(* alternatively
Sched.nDefaultValue										:= E_BA_BuildingMode.eDefault;
Sched.bWriteWeekly										:= FALSE;
//	Monday
Sched.aWeek[E_BA_Weekday.eMonday,1].eState				:= E_BA_SchedEntryState.eValue;
Sched.aWeek[E_BA_Weekday.eMonday,1].uValue.udiVal		:= E_BA_BuildingMode.eCleaning;
Sched.aWeek[E_BA_Weekday.eMonday,1].stTime.nHour		:= 19;
Sched.aWeek[E_BA_Weekday.eMonday,1].stTime.nMinute		:= 0;
Sched.aWeek[E_BA_Weekday.eMonday,1].stTime.nSecond		:= 0;
Sched.aWeek[E_BA_Weekday.eMonday,2].eState				:= E_BA_SchedEntryState.eValue;
Sched.aWeek[E_BA_Weekday.eMonday,2].uValue.udiVal		:= E_BA_BuildingMode.eNightWatch;
Sched.aWeek[E_BA_Weekday.eMonday,2].stTime.nHour		:= 20;
Sched.aWeek[E_BA_Weekday.eMonday,2].stTime.nMinute		:= 0;
Sched.aWeek[E_BA_Weekday.eMonday,2].stTime.nSecond		:= 0;
Sched.aWeek[E_BA_Weekday.eMonday,3].eState				:= E_BA_SchedEntryState.eValue;
Sched.aWeek[E_BA_Weekday.eMonday,3].uValue.udiVal		:= E_BA_BuildingMode.eDefault;
Sched.aWeek[E_BA_Weekday.eMonday,3].stTime.nHour		:= 0;
Sched.aWeek[E_BA_Weekday.eMonday,3].stTime.nMinute		:= 0;
Sched.aWeek[E_BA_Weekday.eMonday,3].stTime.nSecond		:= 0;
//	Tuesday
Sched.aWeek[E_BA_Weekday.eTuesday,1].eState				:= E_BA_SchedEntryState.eValue;
Sched.aWeek[E_BA_Weekday.eTuesday,1].uValue.udiVal		:= E_BA_BuildingMode.eCleaning;
Sched.aWeek[E_BA_Weekday.eTuesday,1].stTime.nHour		:= 19;
Sched.aWeek[E_BA_Weekday.eTuesday,1].stTime.nMinute		:= 0;
Sched.aWeek[E_BA_Weekday.eTuesday,1].stTime.nSecond		:= 0;
Sched.aWeek[E_BA_Weekday.eTuesday,2].eState				:= E_BA_SchedEntryState.eValue;
Sched.aWeek[E_BA_Weekday.eTuesday,2].uValue.udiVal		:= E_BA_BuildingMode.eNightWatch;
Sched.aWeek[E_BA_Weekday.eTuesday,2].stTime.nHour		:= 20;
Sched.aWeek[E_BA_Weekday.eTuesday,2].stTime.nMinute		:= 0;
Sched.aWeek[E_BA_Weekday.eTuesday,2].stTime.nSecond		:= 0;
Sched.aWeek[E_BA_Weekday.eTuesday,3].eState				:= E_BA_SchedEntryState.eValue;
Sched.aWeek[E_BA_Weekday.eTuesday,3].uValue.udiVal		:= E_BA_BuildingMode.eDefault;
Sched.aWeek[E_BA_Weekday.eTuesday,3].stTime.nHour		:= 0;
Sched.aWeek[E_BA_Weekday.eTuesday,3].stTime.nMinute		:= 0;
Sched.aWeek[E_BA_Weekday.eTuesday,3].stTime.nSecond		:= 0;
//	Wednesday
Sched.aWeek[E_BA_Weekday.eWednesday,1].eState			:= E_BA_SchedEntryState.eValue;
Sched.aWeek[E_BA_Weekday.eWednesday,1].uValue.udiVal	:= E_BA_BuildingMode.eCleaning;
Sched.aWeek[E_BA_Weekday.eWednesday,1].stTime.nHour		:= 19;
Sched.aWeek[E_BA_Weekday.eWednesday,1].stTime.nMinute	:= 0;
Sched.aWeek[E_BA_Weekday.eWednesday,1].stTime.nSecond	:= 0;
Sched.aWeek[E_BA_Weekday.eWednesday,2].eState			:= E_BA_SchedEntryState.eValue;
Sched.aWeek[E_BA_Weekday.eWednesday,2].uValue.udiVal	:= E_BA_BuildingMode.eNightWatch;
Sched.aWeek[E_BA_Weekday.eWednesday,2].stTime.nHour		:= 20;
Sched.aWeek[E_BA_Weekday.eWednesday,2].stTime.nMinute	:= 0;
Sched.aWeek[E_BA_Weekday.eWednesday,2].stTime.nSecond	:= 0;
Sched.aWeek[E_BA_Weekday.eWednesday,3].eState			:= E_BA_SchedEntryState.eValue;
Sched.aWeek[E_BA_Weekday.eWednesday,3].uValue.udiVal	:= E_BA_BuildingMode.eDefault;
Sched.aWeek[E_BA_Weekday.eWednesday,3].stTime.nHour		:= 0;
Sched.aWeek[E_BA_Weekday.eWednesday,3].stTime.nMinute	:= 0;
Sched.aWeek[E_BA_Weekday.eWednesday,3].stTime.nSecond	:= 0;
//	Thursday
Sched.aWeek[E_BA_Weekday.eThursday,1].eState			:= E_BA_SchedEntryState.eValue;
Sched.aWeek[E_BA_Weekday.eThursday,1].uValue.udiVal		:=E_BA_BuildingMode.eCleaning;
Sched.aWeek[E_BA_Weekday.eThursday,1].stTime.nHour		:= 19;
Sched.aWeek[E_BA_Weekday.eThursday,1].stTime.nMinute	:= 0;
Sched.aWeek[E_BA_Weekday.eThursday,1].stTime.nSecond	:= 0;
Sched.aWeek[E_BA_Weekday.eThursday,2].eState			:= E_BA_SchedEntryState.eValue;
Sched.aWeek[E_BA_Weekday.eThursday,2].uValue.udiVal		:= E_BA_BuildingMode.eNightWatch;
Sched.aWeek[E_BA_Weekday.eThursday,2].stTime.nHour		:= 20;
Sched.aWeek[E_BA_Weekday.eThursday,2].stTime.nMinute	:= 0;
Sched.aWeek[E_BA_Weekday.eThursday,2].stTime.nSecond	:= 0;
Sched.aWeek[E_BA_Weekday.eThursday,3].eState			:= E_BA_SchedEntryState.eValue;
Sched.aWeek[E_BA_Weekday.eThursday,3].uValue.udiVal		:= E_BA_BuildingMode.eDefault;
Sched.aWeek[E_BA_Weekday.eThursday,3].stTime.nHour		:= 0;
Sched.aWeek[E_BA_Weekday.eThursday,3].stTime.nMinute	:= 0;
Sched.aWeek[E_BA_Weekday.eThursday,3].stTime.nSecond	:= 0;
//	Friday
Sched.aWeek[E_BA_Weekday.eFriday,1].eState				:= E_BA_SchedEntryState.eValue;
Sched.aWeek[E_BA_Weekday.eFriday,1].uValue.udiVal		:= E_BA_BuildingMode.eCleaning;
Sched.aWeek[E_BA_Weekday.eFriday,1].stTime.nHour		:= 19;
Sched.aWeek[E_BA_Weekday.eFriday,1].stTime.nMinute		:= 0;
Sched.aWeek[E_BA_Weekday.eFriday,1].stTime.nSecond		:= 0;
Sched.aWeek[E_BA_Weekday.eFriday,2].eState				:= E_BA_SchedEntryState.eValue;
Sched.aWeek[E_BA_Weekday.eFriday,2].uValue.udiVal		:= E_BA_BuildingMode.eNightWatch;
Sched.aWeek[E_BA_Weekday.eFriday,2].stTime.nHour		:= 20;
Sched.aWeek[E_BA_Weekday.eFriday,2].stTime.nMinute		:= 0;
Sched.aWeek[E_BA_Weekday.eFriday,2].stTime.nSecond		:= 0;
Sched.aWeek[E_BA_Weekday.eFriday,3].eState				:= E_BA_SchedEntryState.eValue;
Sched.aWeek[E_BA_Weekday.eFriday,3].uValue.udiVal		:= E_BA_BuildingMode.eDefault;
Sched.aWeek[E_BA_Weekday.eFriday,3].stTime.nHour		:= 0;
Sched.aWeek[E_BA_Weekday.eFriday,3].stTime.nMinute		:= 0;
Sched.aWeek[E_BA_Weekday.eFriday,3].stTime.nSecond		:= 0; 
*)
END_METHOD

END_FUNCTION_BLOCK

// ---- Templates/POUs/Trade/BuildingAutomation/GlobalEventsAndSettings/FB_BA_WeatherParameter.TcPOU
{region '#Template'}
	{attribute 'Version' := '5.0.0.0'}
	{attribute 'Tags' := '"LCID": "1031", "Text": "General, Settings, Parameters, Basics"'}
	{attribute 'Tags' := '"LCID": "1033", "Text": "General, Settings, Parameters, Basics"'}
	{attribute 'Using' := '"Type": "Template", "URI": "BA2_Param"'}
	{attribute 'Description' := '"LCID": "1031", "Text": "Witterungsparameter für die Templates"'}
	{attribute 'Description' := '"LCID": "1033", "Text": "Weather parameters for the templates"'}
{endregion}
FUNCTION_BLOCK FB_BA_WeatherParameter EXTENDS FB_BA_View
VAR_INPUT
	fTWth					: REAL;	//	Weather temperature
END_VAR
VAR_OUTPUT
	fSpFrstProtec			: REAL;  // frost protection setpoint. for eg. Heating circutis in protection mode
	fTWthLowLimit			: REAL;  // below this value all frostprotection funcktions in HVAC-Plants will be enabled
	bTWthLowLimit			: BOOL;  // is TRUE when the outside temperature is below the value from fTWthLowLimit 
	fTWthDamped				: REAL;  // damped outside temperature
	bTWthDampedLowLimit		: BOOL;	
END_VAR
VAR_INPUT CONSTANT
	SpFrstProtec			: FB_BA_AV_Op;		
	TWthLowLimitVal			: FB_BA_AV_Op;																
	TWthLowLimit			: FB_BA_BV_Op;								
	TWthDamped				: FB_BA_AV_Op;		
	TWthDampedLowLimit		: FB_BA_BV_Op;	
END_VAR
VAR
	TWthLowLimitHys			: FB_BA_Swi2P;
	Average					: FB_BA_TiAvrg;
	TWthDampedLowLimitHys	: FB_BA_Swi2P;
END_VAR

SUPER^(); // FB_BA_View
SpFrstProtec(); // FB_BA_AV_Op
fSpFrstProtec := SpFrstProtec.fPresentValue;
TWthLowLimitVal(); // FB_BA_AV_Op
fTWthLowLimit := TWthLowLimitVal.fPresentValue;
TWthLowLimitHys(bEn := TRUE, fIn := fTWth, fOn := fTWthLowLimit, fOff := fTWthLowLimit + 1); // FB_BA_Swi2P
TWthLowLimit(bValuePgm := TWthLowLimitHys.bQ); // FB_BA_BV_Op
bTWthLowLimit := TWthLowLimit.bPresentValue;
Average(bEn := BA2_Param.bDlyStartPLC, fIn := fTWth, nIntval := 900, nNumOfElem := 96); // FB_BA_TiAvrg
TWthDamped(fValuePgm := Average.fOut); // FB_BA_AV_Op
fTWthDamped := TWthDamped.fPresentValue;
TWthDampedLowLimitHys(bEn := TRUE, fIn := fTWthDamped, fOn := fTWthLowLimit, fOff := fTWthLowLimit + 1.0); // FB_BA_Swi2P
TWthDampedLowLimit(bValuePgm := TWthDampedLowLimitHys.bQ); // FB_BA_BV_Op
bTWthDampedLowLimit := TWthDampedLowLimit.bPresentValue;

METHOD FB_init : BOOL
VAR_INPUT
	bInitRetains : BOOL; // if TRUE, the retain variables are initialized (warm start / cold start)
	bInCopyCode : BOOL;  // if TRUE, the instance afterwards gets moved into the copy code (online change)
END_VAR
SpFrstProtec.iParent				:= THIS^;
SpFrstProtec.iLabel					:= LblCtl_SetpointFrostProtection;
SpFrstProtec.eUnit					:= E_BA_Unit.eTemperature_DegreesCelsius;  
SpFrstProtec.fValueRm				:= 5.0;
SpFrstProtec.fCOVIncrement			:= BA2_Param.fDefCOVIncrement;							

TWthLowLimitVal.iParent				:= THIS^;
TWthLowLimitVal.iLabel				:= LblCtl_SetpointMinimumOutsideTemperature;
TWthLowLimitVal.eUnit				:= E_BA_Unit.eTemperature_DegreesCelsius;  
TWthLowLimitVal.fValueRm			:= 8.0;
TWthLowLimitVal.fCOVIncrement		:= BA2_Param.fDefCOVIncrement;							

TWthLowLimit.iParent				:= THIS^;	
TWthLowLimit.iLabel					:= LblCtl_OperationalMessageTemperatureWeatherLowLimit;
TWthLowLimit.sInactiveText			:= txtEvent_Off;
TWthLowLimit.sActiveText			:= txtEvent_On;
TWthLowLimit.bValueRm				:= FALSE;		
TWthLowLimit.eToggleMode 			:= E_BA_ToggleMode.eSwitch;

TWthDamped.iParent					:= THIS^;
TWthDamped.iLabel					:= LblCtl_MeanDamped;
TWthDamped.eUnit					:= E_BA_Unit.eTemperature_DegreesCelsius;  
TWthDamped.fValueRm					:= 0.0;
TWthDamped.fCOVIncrement			:= BA2_Param.fDefCOVIncrement;							

TWthDampedLowLimit.iParent			:= THIS^;	
TWthDampedLowLimit.iLabel			:= LblCtl_OperationalMessageTemperatureWeatherDampedLowLimit;	
TWthDampedLowLimit.sInactiveText	:= txtEvent_Off;
TWthDampedLowLimit.sActiveText		:= txtEvent_On;
TWthDampedLowLimit.bValueRm			:= FALSE;								
TWthDampedLowLimit.eToggleMode 		:= E_BA_ToggleMode.eSwitch;
END_METHOD

END_FUNCTION_BLOCK

// ---- Templates/POUs/Trade/BuildingAutomation/WeatherStation/FB_BA_WeatherStation_Draft.TcPOU
{region '#Template'}
	{attribute 'Version' := '5.0.1.0'}
	{attribute 'Tags' := '"LCID": "1031", "Text": "Plant, Weatherstation, Draft"'}
	{attribute 'Tags' := '"LCID": "1033", "Text": "Plant, Weatherstation, Draft"'}
	{attribute 'Using' := '"Type": "Template", "URI": "LblComp"'}		 		 
	{attribute 'Description' := '"LCID": "1031", "Text": "Vorlage-Template: beinhaltet alle Objekte, die Eingangsverknüpfung zu diesen muss vom Anwender erstellt werden"'}
	{attribute 'Description' := '"LCID": "1033", "Text": "Draft-template: contains all objects to be connected to appropriate inputs by the user"'}
{endregion}
FUNCTION_BLOCK FB_BA_WeatherStation_Draft EXTENDS FB_BA_View
VAR_INPUT CONSTANT
	Dstb						: FB_BA_BI;
	Rain						: FB_BA_BI;
	WthT						: FB_BA_AI;
	DewPtT						: FB_BA_AI; 
	PrssAbs						: FB_BA_AI;
	PrssRel						: FB_BA_AI;
	HumAbs						: FB_BA_AI;
	HumRel						: FB_BA_AI;
	Brightness_N				: FB_BA_AI;
	Brightness_S				: FB_BA_AI;
	Brightness_E				: FB_BA_AI;
	Brightness_W				: FB_BA_AI;
	Dawn						: FB_BA_AI;
	GlobRadn					: FB_BA_AI;      
	WndDir						: FB_BA_AI;
	WndSpd						: FB_BA_AI; 
	Latd						: FB_BA_AI;  
	Lngt						: FB_BA_AI; 
	SunAzm						: FB_BA_AI;
	SunElv						: FB_BA_AI;                 
END_VAR	

VAR
	stDateTime_PLACEHOLDER		: TIMESTRUCT;			// Placeholder-variable, so the template can be compiled correctly
														// to be replaced by an appropriate timestruct
END_VAR

SUPER^(); // FB_BA_View
Dstb(); // FB_BA_BI
Site.stWeatherStation.bDisturb := Dstb.bPresentValue;
Rain(); // FB_BA_BI
Site.stWeatherStation.bRain := Rain.bPresentValue;
WndSpd(); // FB_BA_AI
Site.stWeatherStation.fWindSpeed := WndSpd.fPresentValue;
WthT(); // FB_BA_AI
Site.stWeatherStation.fOutsideTemperature := WthT.fPresentValue;
DewPtT(); // FB_BA_AI
Site.stWeatherStation.fDewPointTemperature := DewPtT.fPresentValue;
PrssAbs(); // FB_BA_AI
Site.stWeatherStation.fPressureAbs := PrssAbs.fPresentValue;
PrssRel(); // FB_BA_AI
Site.stWeatherStation.fPressureRel := PrssRel.fPresentValue;
Dawn(); // FB_BA_AI
Site.stWeatherStation.fDawn := Dawn.fPresentValue;
GlobRadn(); // FB_BA_AI
Site.stWeatherStation.fGlobalRadiation := GlobRadn.fPresentValue;
WndDir(); // FB_BA_AI
Site.stWeatherStation.fWindDirection := WndDir.fPresentValue;
HumAbs(); // FB_BA_AI
Site.stWeatherStation.fHumidityAbs := HumAbs.fPresentValue;
HumRel(); // FB_BA_AI
Site.stWeatherStation.fHumidityRel := HumRel.fPresentValue;
Latd(); // FB_BA_AI
Site.stWeatherStation.fLatitude := Latd.fPresentValue;
Lngt(); // FB_BA_AI
Site.stWeatherStation.fLongitude := Lngt.fPresentValue;
SunAzm(); // FB_BA_AI
Site.stWeatherStation.fSunAzimuth := SunAzm.fPresentValue;
SunElv(); // FB_BA_AI
Site.stWeatherStation.fSunElevation := SunElv.fPresentValue;
Brightness_N(); // FB_BA_AI
Site.stWeatherStation.fBrightnessNorth := Brightness_N.fPresentValue;
Brightness_S(); // FB_BA_AI
Site.stWeatherStation.fBrightnessSouth := Brightness_S.fPresentValue;
Brightness_E(); // FB_BA_AI
Site.stWeatherStation.fBrightnessEast := Brightness_E.fPresentValue;
Brightness_W(); // FB_BA_AI
Site.stWeatherStation.fBrightnessWest := Brightness_W.fPresentValue;
Site.stWeatherStation.stDateTime := stDateTime_PLACEHOLDER;

METHOD FB_init : BOOL
VAR_INPUT
	bInitRetains : BOOL; // if TRUE, the retain variables are initialized (warm start / cold start)
	bInCopyCode : BOOL;  // if TRUE, the instance afterwards gets moved into the copy code (online change)
END_VAR
Dstb.iParent							:= THIS^;
Dstb.iLabel								:= LblComp_Wth_WeatherStation; 	
Dstb.sActiveText 						:= txtEvent_Yes;
Dstb.sInactiveText 						:= txtEvent_No;
Dstb.nEventClassID						:= EC_ID.NC60;
Dstb.aEventTransitionText[1]			:= txtEvent_No;
Dstb.aEventTransitionText[2]			:= txtEvent_None;
Dstb.aEventTransitionText[3]			:= txtEvent_Yes;
Dstb.bEventDetectionEnable				:= FALSE;	  
						
Rain.iParent							:= THIS^;
Rain.iLabel								:= LblComp_Wth_RainSensor; 	
Rain.sActiveText 						:= txtEvent_Yes;
Rain.sInactiveText 						:= txtEvent_No;
Rain.nEventClassID						:= EC_ID.NC60;
Rain.aEventTransitionText[1]			:= txtEvent_No;
Rain.aEventTransitionText[2]			:= txtEvent_None;
Rain.aEventTransitionText[3]			:= txtEvent_Yes;
Rain.bEventDetectionEnable				:= FALSE;	
						
WthT.iParent							:= THIS^;
WthT.iLabel								:= LblComp_Wth_TemperatureOutside; 	
WthT.eUnit 								:= E_BA_Unit.eTemperature_DegreesCelsius;	
WthT.nEventClassID						:= EC_ID.NC40;
										
DewPtT.iParent							:= THIS^;
DewPtT.iLabel							:= LblComp_Wth_TemperatureDewPoint; 		
DewPtT.eUnit							:= E_BA_Unit.eTemperature_DegreesCelsius;
DewPtT.nEventClassID					:= EC_ID.NC40;
						
PrssAbs.iParent							:= THIS^;
PrssAbs.iLabel							:= LblComp_Wth_PressureAbsolute; 
PrssAbs.eUnit							:= E_BA_Unit.ePressure_Hectopascals;
PrssAbs.nEventClassID					:= EC_ID.NC40;
										
PrssRel.iParent							:= THIS^;
PrssRel.iLabel							:= LblComp_Wth_PressureRelative; 	
PrssRel.eUnit							:= E_BA_Unit.ePressure_Hectopascals;
PrssRel.nEventClassID					:= EC_ID.NC40;
						
HumAbs.iParent							:= THIS^;
HumAbs.iLabel							:= LblComp_Wth_AbsoluteHumidityOutsideAir; 
HumAbs.eUnit							:= E_BA_Unit.eHumidity_GramsOfWaterPerKilogramDryAir;
HumAbs.nEventClassID					:= EC_ID.NC40;
										
HumRel.iParent							:= THIS^;
HumRel.iLabel							:= LblComp_Wth_RelativeHumidityOutsideAir; 
HumRel.eUnit							:= E_BA_Unit.eHumidity_PercentRelativeHumidity;
HumRel.nEventClassID					:= EC_ID.NC40;
						
Brightness_N.iParent					:= THIS^;
Brightness_N.iLabel						:= LblComp_Wth_Brightness; 		
Brightness_N.eUnit						:= E_BA_Unit.eLight_Luxes;
Brightness_N.nEventClassID				:= EC_ID.NC40;
                                        
Brightness_S.iParent					:= THIS^;
Brightness_S.iLabel						:= LblComp_Wth_Brightness; 		
Brightness_S.eUnit						:= E_BA_Unit.eLight_Luxes;
Brightness_S.nEventClassID				:= EC_ID.NC40;
                                        
Brightness_E.iParent					:= THIS^;
Brightness_E.iLabel						:= LblComp_Wth_Brightness; 		
Brightness_E.eUnit						:= E_BA_Unit.eLight_Luxes;
Brightness_E.nEventClassID				:= EC_ID.NC40;
                                        
Brightness_W.iParent					:= THIS^;
Brightness_W.iLabel						:= LblComp_Wth_Brightness; 		
Brightness_W.eUnit						:= E_BA_Unit.eLight_Luxes;
Brightness_W.nEventClassID				:= EC_ID.NC40;

Dawn.iParent							:= THIS^;
Dawn.iLabel								:= LblComp_Wth_Dawn; 	
Dawn.eUnit								:= E_BA_Unit.eLight_Luxes;
Dawn.nEventClassID						:= EC_ID.NC40;
						
GlobRadn.iParent						:= THIS^;
GlobRadn.iLabel							:= LblComp_Wth_SolarRadiation; 	
GlobRadn.eUnit							:= E_BA_Unit.eLight_WattsPerSquareMeter;
GlobRadn.nEventClassID					:= EC_ID.NC40;
						
WndDir.iParent							:= THIS^;
WndDir.iLabel							:= LblComp_Wth_WindDirection; 	
WndDir.eUnit							:= E_BA_Unit.eOther_DegreesAngular;
WndDir.nEventClassID					:= EC_ID.NC40;
										
WndSpd.iParent							:= THIS^;
WndSpd.iLabel							:= LblComp_Wth_WindSpeed; 	
WndSpd.eUnit							:= E_BA_Unit.eVelocity_MetersPerSecond;
WndSpd.nEventClassID					:= EC_ID.NC40;
						
Latd.iParent							:= THIS^;
Latd.iLabel								:= LblComp_Wth_GeoLatitude; 	
Latd.eUnit								:= E_BA_Unit.eOther_DegreesAngular;
Latd.nEventClassID						:= EC_ID.NC40;
										
Lngt.iParent							:= THIS^;
Lngt.iLabel								:= LblComp_Wth_GeoLongitude; 	
Lngt.eUnit								:= E_BA_Unit.eOther_DegreesAngular;
Lngt.nEventClassID						:= EC_ID.NC40;
						
SunAzm.iParent							:= THIS^;
SunAzm.iLabel							:= LblComp_Wth_SunAzimuth; 	
SunAzm.eUnit							:= E_BA_Unit.eOther_DegreesAngular;
SunAzm.nEventClassID					:= EC_ID.NC40;
						
SunElv.iParent							:= THIS^;
SunElv.iLabel							:= LblComp_Wth_SunElevation; 	
SunElv.eUnit							:= E_BA_Unit.eOther_DegreesAngular;
SunElv.nEventClassID					:= EC_ID.NC40;
END_METHOD

END_FUNCTION_BLOCK

// ---- Templates/POUs/Trade/BuildingAutomation/Communication/FB_BA_AdsComServer.TcPOU
{region '#Template'}
	{attribute 'Version' := '5.0.0.0'}
	{attribute 'Tags' := '"LCID": "1031", "Text": "Gebäudeautomation, Kommunikation, Server, Client, Publisher, Subscriber"'}
	{attribute 'Tags' := '"LCID": "1033", "Text": "Building automation, Communication, Server, Client, Publisher, Subscriber"'}
	{attribute 'Using' := '"Type": "Template", "URI": "Site"'}
	{attribute 'Description' := '"LCID": "1031", "Text": "Server Datenkommunikation"'}
	{attribute 'Description' := '"LCID": "1033", "Text": "Server data communication"'}
{endregion}

FUNCTION_BLOCK FB_BA_AdsComServer
VAR_INPUT
END_VAR
VAR_OUTPUT
END_VAR
VAR_INPUT CONSTANT
	WeatherStation					: FB_BA_RawPublisher;			
	GeneralSettings					: FB_BA_RawPublisher;												
END_VAR
VAR
END_VAR

GeneralSettings(xData := Site.stGeneralSettings); // FB_BA_RawPublisher
WeatherStation(xData := Site.stWeatherStation); // FB_BA_RawPublisher

END_FUNCTION_BLOCK

// ---- Templates/POUs/Trade/AirConditioning/FB_BA_AirConditioning.TcPOU
{region '#Template'}
	{attribute 'Version' := '5.0.0.0'}
	{attribute 'Tags' := '"LCID": "1031", "Text": "Trade, Plant, AC"'}
	{attribute 'Tags' := '"LCID": "1033", "Text": "Trade, Plant, AC"'}
	{attribute 'Using' := '"Type": "Template", "URI": "Priority"'}		 		 
	{attribute 'Using' := '"Type": "Template", "URI": "Site"'}
	{attribute 'Description' := '"LCID": "1031", "Text": "Aufruf der Anlagen des Gewerks Klimaanlagen"'}
	{attribute 'Description' := '"LCID": "1033", "Text": "Calling the plants of the trade air conditioning"'}
{endregion}
FUNCTION_BLOCK FB_BA_AirConditioning EXTENDS FB_BA_View
VAR_INPUT CONSTANT
	AHU01				: FB_BA_AHU_1st_10;
END_VAR
VAR_INPUT
END_VAR
VAR_OUTPUT
END_VAR
VAR
END_VAR

SUPER^(); // FB_BA_View
AHU01(); // FB_BA_AHU_1st_10

METHOD FB_init : BOOL
VAR_INPUT
	bInitRetains : BOOL; // if TRUE, the retain variables are initialized (warm start / cold start)
	bInCopyCode : BOOL;  // if TRUE, the instance afterwards gets moved into the copy code (online change)
END_VAR
AHU01.iParent 				:= THIS^;	
AHU01.iLabel				:= LblPlt_Partial_air_conditioning_system;	
AHU01.sObjectName			:= '{Idx=01}';  
AHU01.eDPADMode				:= E_BA_DPADMode.eInclude;
END_METHOD

END_FUNCTION_BLOCK

// ---- Templates/POUs/Trade/HeatingSystem/FB_BA_Heating.TcPOU
{region '#Template'}
	{attribute 'Version' := '5.0.0.0'}
	{attribute 'Tags' := '"LCID": "1031", "Text": "Trade, Plant, Heating System"'}
	{attribute 'Tags' := '"LCID": "1033", "Text": "Trade, Plant, Heating System"'}
	{attribute 'Using' := '"Type": "Template", "URI": "Site"'}
	{attribute 'Description' := '"LCID": "1031", "Text": "Aufruf der Anlagen des Gewerks Heizsysteme"'}
	{attribute 'Description' := '"LCID": "1033", "Text": "Calling the plants of the trade heating system"'}
{endregion}
FUNCTION_BLOCK FB_BA_Heating EXTENDS FB_BA_View
VAR_INPUT CONSTANT
	HTC01				: FB_BA_H_HtgCir01;		
END_VAR
VAR_INPUT
END_VAR
VAR_OUTPUT
END_VAR
VAR
END_VAR

SUPER^(); // FB_BA_View
HTC01(); // FB_BA_H_HtgCir01

METHOD FB_init : BOOL
VAR_INPUT
	bInitRetains : BOOL; // if TRUE, the retain variables are initialized (warm start / cold start)
	bInCopyCode : BOOL;  // if TRUE, the instance afterwards gets moved into the copy code (online change)
END_VAR
HTC01.iParent 					:= THIS^;	
HTC01.iLabel						:= LblPlt_Heating_circuit;	
HTC01.sObjectName				:= '{Idx=01}';  
HTC01.eDPADMode					:= E_BA_DPADMode.eInclude;
END_METHOD

END_FUNCTION_BLOCK

// ---- Templates/POUs/Trade/RoomAutomation/FB_BA_RoomAutomation.TcPOU
{region '#Template'}
	{attribute 'Version' := '5.0.0.0'}
	{attribute 'Tags' := '"LCID": "1031", "Text": "Trade, Plant, Room automation"'}
	{attribute 'Tags' := '"LCID": "1033", "Text": "Trade, Plant, Room automation"'}
	{attribute 'Using' := '"Type": "Template", "URI": "Site"'}
	{attribute 'Description' := '"LCID": "1031", "Text": "Aufruf der Anlagen des Gewerks Raumautomation"'}
	{attribute 'Description' := '"LCID": "1033", "Text": "Calling the plants of the trade room automation"'}
{endregion}
FUNCTION_BLOCK FB_BA_RoomAutomation EXTENDS FB_BA_View
VAR_INPUT CONSTANT
//	RoomGeneral		: FB_BA_RoomGeneral	;
//	SampleRoom		: FB_BA_RoomSample1;			
END_VAR

SUPER^(); // FB_BA_View

METHOD FB_init : BOOL
VAR_INPUT
	bInitRetains : BOOL; // if TRUE, the retain variables are initialized (warm start / cold start)
	bInCopyCode : BOOL;  // if TRUE, the instance afterwards gets moved into the copy code (online change)
END_VAR
// RoomGeneral.iParent			:= THIS^;
// RoomGeneral.sObjectName		:= '{RAU{Idx=01}}';
// RoomGeneral.sDescription		:= 'Room automation';
// RoomGeneral.eDPADMode		:= E_BA_DPADMode.eInclude;

// SampleRoom.iParent			:= THIS^;	
// SampleRoom.sObjectName		:= '{SRO{Idx=01}}';
// SampleRoom.sDescription		:= 	'Sample room'; 	
// SampleRoom.eDPADMode			:= E_BA_DPADMode.eInclude;
END_METHOD

END_FUNCTION_BLOCK

// ---- Templates/POUs/Trade/AutomationControl/Device/TimeSettings/FB_BA_BACnetTime_TO_SysTime.TcPOU
{region '#Template'}
	{attribute 'Version' := '5.0.1.0'}
	{attribute 'Tags' := '"LCID": "1031", "Text": "Automatisierungssteuerung, Gerät, Einstellungen, Systemzeit, BACnet Adapter Zeit"'}
	{attribute 'Tags' := '"LCID": "1033", "Text": "Automation control, Device, Settings, Systemzeit, BACnet Adapter Time"'}
	{attribute 'Using' := '"Type": "Template", "URI": "SysTime"'}		 		 
	{attribute 'Description' := '"LCID": "1031", "Text": "BACnet Adapter Zeit abrufen und lokal setzen"'}
	{attribute 'Description' := '"LCID": "1033", "Text": "Get BACnet Adapter Time and set locally"'}
{endregion}

FUNCTION_BLOCK FB_BA_BACnetTime_TO_SysTime
VAR_INPUT
END_VAR
VAR_OUTPUT
END_VAR
VAR_INPUT CONSTANT PERSISTENT	
	sExternalAmsNetId						: T_AmsNetId := ''; // Beispiel,Example: '192.168.131.1.1.1'
	{attribute 'parameterUnit':= 's'}
	GetLocalSysTime_nTiAuto					: UDINT := 60;
END_VAR	
VAR_INPUT CONSTANT
	GetExtSysTime				: FB_BA_GetTime;

	SetSysTimeLocal				: FB_BA_SetTime;

	GetLocalSysTime				: FB_BA_GetTime;
	GetBACnetAdapterTime		: FB_BACnet_GetAdapterTime;
END_VAR
VAR
	GetExtSysTime_bSync					: BOOL;	
	GetExtSysTime_rtrigSync				: R_TRIG;
	
	GetBACnetAdapterTime_wYear				: WORD;
	GetBACnetAdapterTime_wMonth				: WORD;
	GetBACnetAdapterTime_wDayOfWeek			: WORD;
	GetBACnetAdapterTime_wDay				: WORD;
	GetBACnetAdapterTime_wHour				: WORD;
	GetBACnetAdapterTime_wMinute			: WORD;
	GetBACnetAdapterTime_wSecond			: WORD;
	GetBACnetAdapterTime_wMilliseconds		: WORD;		
	
	// F_BA_STDateTime_TO_TIMESTRUCT
END_VAR

GetBACnetAdapterTime(); // FB_BACnet_GetAdapterTime
GetBACnetAdapterTime_wYear := GetBACnetAdapterTime.stTimeStruct.TIMESTRUCT;
GetBACnetAdapterTime_wMonth := GetBACnetAdapterTime.stTimeStruct.wYear;
GetBACnetAdapterTime_wDayOfWeek := GetBACnetAdapterTime.stTimeStruct.wMonth;
GetBACnetAdapterTime_wDay := GetBACnetAdapterTime.stTimeStruct.wDayOfWeek;
GetBACnetAdapterTime_wHour := GetBACnetAdapterTime.stTimeStruct.wDay;
GetBACnetAdapterTime_wMinute := GetBACnetAdapterTime.stTimeStruct.wHour;
GetBACnetAdapterTime_wSecond := GetBACnetAdapterTime.stTimeStruct.wMinute;
GetBACnetAdapterTime_wMilliseconds := GetBACnetAdapterTime.stTimeStruct.wSecond;
SetSysTimeLocal(
    bSet := GetBACnetAdapterTime.bSuccess,
    tNetId := '',
    tSysTi := GetBACnetAdapterTime.stTimeStruct); // FB_BA_SetTime
GetLocalSysTime(bEn := TRUE, tNetId := '', nUpdRtc := GetLocalSysTime_nTiAuto); // FB_BA_GetTime
SysTime.stSystemTime := GetLocalSysTime.tSysTi;
SysTime.stSystemTimeUTC := GetLocalSysTime.tUTC;
SysTime.dtSystemTime := GetLocalSysTime.dtSysTi;
SysTime.dtSystemTimeUTC := GetLocalSysTime.dtUTC;

END_FUNCTION_BLOCK

// ---- Templates/POUs/Trade/AutomationControl/Device/TimeSettings/FB_BA_ExternalSysTime.TcPOU
{region '#Template'}
	{attribute 'Version' := '5.0.0.0'}
	{attribute 'Tags' := '"LCID": "1031", "Text": "Automatisierungssteuerung, Gerät, Einstellungen, Systemzeit, BACnet Adapter Time"'}
	{attribute 'Tags' := '"LCID": "1033", "Text": "Automation control, Device, Settings, Systemzeit, BACnet Adapter Zeit"'}
	{attribute 'Using' := '"Type": "Template", "URI": "SysTime"'}		 		 
	{attribute 'Description' := '"LCID": "1031", "Text": "Externe Systemzeit abrufen und lokal setzen"'}
	{attribute 'Description' := '"LCID": "1033", "Text": "Get external system time and set locally"'}
{endregion}

FUNCTION_BLOCK FB_BA_ExternalSysTime
VAR_INPUT
END_VAR
VAR_OUTPUT
END_VAR
VAR_INPUT CONSTANT PERSISTENT	
	sExternalAmsNetId						: T_AmsNetId := ''; // Beispiel,Example: '192.168.131.1.1.1'
	{attribute 'parameterUnit':= 's'}
	GetExtSysTime_nTiAuto					: UDINT := 600;
	{attribute 'parameterUnit':= 's'}
	GetLocalSysTime_nTiAuto					: UDINT := 60;
END_VAR	
VAR_INPUT CONSTANT
	GetExtSysTime				: FB_BA_GetTime;

	SetSysTimeLocal				: FB_BA_SetTime;
	SetBACnetAdapterTime		: FB_BA_SetBACnetAdapterTime;

	GetLocalSysTime				: FB_BA_GetTime;
	GetBACnetAdapterTime		: FB_BA_GetBACnetAdapterTime;
END_VAR
VAR
	GetExtSysTime_bSync					: BOOL;	
	GetExtSysTime_rtrigSync				: R_TRIG;
	
	GetBACnetAdapterTime_wYear				: WORD;
	GetBACnetAdapterTime_wMonth				: WORD;
	GetBACnetAdapterTime_wDayOfWeek			: WORD;
	GetBACnetAdapterTime_wDay				: WORD;
	GetBACnetAdapterTime_wHour				: WORD;
	GetBACnetAdapterTime_wMinute			: WORD;
	GetBACnetAdapterTime_wSecond			: WORD;
	GetBACnetAdapterTime_wMilliseconds		: WORD;		
	
	// F_BA_STDateTime_TO_TIMESTRUCT
END_VAR

GetExtSysTime(bEn := TRUE, tNetId := sExternalAmsNetId, nUpdRtc := GetExtSysTime_nTiAuto); // FB_BA_GetTime
GetExtSysTime_rtrigSync(CLK := GetExtSysTime.bRdySysTi); // R_TRIG
GetExtSysTime_bSync := GetExtSysTime_rtrigSync.Q;
SetSysTimeLocal(bSet := GetExtSysTime_bSync, tNetId := '', tSysTi := GetExtSysTime.tSysTi); // FB_BA_SetTime
SetBACnetAdapterTime(bTrig := GetExtSysTime_bSync, stDateTime := F_BA_TIMESTRUCT_TO_DateTime(tValue := GetExtSysTime.tSysTi)); // FB_BA_SetBACnetAdapterTime
GetLocalSysTime(bEn := TRUE, tNetId := '', nUpdRtc := GetLocalSysTime_nTiAuto); // FB_BA_GetTime
SysTime.stSystemTime := GetLocalSysTime.tSysTi;
SysTime.stSystemTimeUTC := GetLocalSysTime.tUTC;
SysTime.dtSystemTime := GetLocalSysTime.dtSysTi;
SysTime.dtSystemTimeUTC := GetLocalSysTime.dtUTC;
GetBACnetAdapterTime(nTiAuto := GetLocalSysTime_nTiAuto); // FB_BA_GetBACnetAdapterTime
GetBACnetAdapterTime_wYear := GetBACnetAdapterTime.stTimeStruct.TIMESTRUCT;
GetBACnetAdapterTime_wMonth := GetBACnetAdapterTime.stTimeStruct.wYear;
GetBACnetAdapterTime_wDayOfWeek := GetBACnetAdapterTime.stTimeStruct.wMonth;
GetBACnetAdapterTime_wDay := GetBACnetAdapterTime.stTimeStruct.wDayOfWeek;
GetBACnetAdapterTime_wHour := GetBACnetAdapterTime.stTimeStruct.wDay;
GetBACnetAdapterTime_wMinute := GetBACnetAdapterTime.stTimeStruct.wHour;
GetBACnetAdapterTime_wSecond := GetBACnetAdapterTime.stTimeStruct.wMinute;
GetBACnetAdapterTime_wMilliseconds := GetBACnetAdapterTime.stTimeStruct.wSecond;

END_FUNCTION_BLOCK

// ---- Templates/POUs/Trade/AirConditioning/Aggregates/Cooler/Temperature/FB_BA_AC_ColTSuACtrl.TcPOU
{region '#Template'}
	{attribute 'Version' := '5.0.1.0'}
	{attribute 'Tags' := '"LCID": "1031", "Text": "AC, Aggregates, Cooler, Temperature, Controller"'}
	{attribute 'Tags' := '"LCID": "1033", "Text": "AC, Aggregates, Cooler, Temperature, Controller"'}
	{attribute 'Using' := '"Type": "Template", "URI": "BA2_Param"'}
	{attribute 'Using' := '"Type": "Template", "URI": "EC_ID"'}
	{attribute 'Using' := '"Type": "Template", "URI": "E_BA_AC_SeqNumber_T"'}
	{attribute 'Description' := '"LCID": "1031", "Text": "Kühler Zuluft Regler Temperatur"'}
	{attribute 'Description' := '"LCID": "1033", "Text": "Cooler Supply air controller temperature"'}
{endregion}
FUNCTION_BLOCK FB_BA_AC_ColTSuACtrl EXTENDS FB_BA_View
VAR_INPUT
	bEn						: BOOL;
	fSpTSuA					: REAL;// Sollwert Temperatur kühlen // Setpoint temperature cooling
	fTSuA					: REAL;// Zuluft Temperatur // Supply air temperature
	bSync					: BOOL;
	fSync					: REAL;
END_VAR
VAR_OUTPUT
	fY              		: REAL;
	bIsActive				: BOOL;	//	active sequence controller
	bSeqActv				: BOOL;	//	Release sequence link, sequence control is active		
END_VAR
VAR_IN_OUT
	stSeqLink				: ST_BA_SeqLink;	//	Sequenz Link Struktur	//	Sequence link structure	
END_VAR
VAR_INPUT CONSTANT
	Ctrl					: FB_BA_SeqCtrl;
END_VAR

SUPER^(); // FB_BA_View
Ctrl(
    bEn := bEn AND stSeqLink.bEnSeqLink,
    fSetpoint := fSpTSuA,
    fCtrlVal := fTSuA,
    eActionPgm := E_BA_Action.eDirect,
    bEnSync := bSync,
    fValSync := fSync,
    nMyNum := E_BA_AC_SeqNumber_T.eCooler,
    stSeqLink := stSeqLink); // FB_BA_SeqCtrl
fY := Ctrl.fPresentValue;
bSeqActv := Ctrl.bSeqActv;
bIsActive := Ctrl.bIsActvSeqCtrl;

METHOD FB_init : BOOL
VAR_INPUT
	bInitRetains : BOOL; // if TRUE, the retain variables are initialized (warm start / cold start)
	bInCopyCode : BOOL;  // if TRUE, the instance afterwards gets moved into the copy code (online change)
END_VAR
Ctrl.iParent						:= THIS^;
Ctrl.iLabel							:= LblFun_LoopObject; 
Ctrl.sObjectName					:= '{Idx=01}';						 
Ctrl.eOpMode						:= E_BA_PIDMode.ePID;								 	 										 	
Ctrl.eOutputUnit					:= E_BA_Unit.eOther_Percent;
Ctrl.fProportionalConstant			:= 3;
Ctrl.fIntegralConstant				:= 180;
Ctrl.fDerivativeConstant			:= 0;
Ctrl.fMaxOutputRm 					:= 100;
Ctrl.fMinOutputRm					:= 0;
Ctrl.fCOVIncrement					:= 0;
Ctrl.nDampConstant					:= 0;
Ctrl.fNeutralZone					:= 0;
END_METHOD

END_FUNCTION_BLOCK

// ---- Templates/POUs/Trade/AirConditioning/Aggregates/ERC/FB_BA_AC_ErcTSuACtrl.TcPOU
{region '#Template'}
	{attribute 'Version' := '5.0.1.0'}
	{attribute 'Tags' := '"LCID": "1031", "Text": "AC, Aggregates, Energy recovery, Temperature, Controller"'}
	{attribute 'Tags' := '"LCID": "1033", "Text": "AC, Aggregates, Energy recovery, Temperature, Controller"'}
	{attribute 'Using' := '"Type": "Template", "URI": "BA2_Param"'}
	{attribute 'Using' := '"Type": "Template", "URI": "EC_ID"'}
	{attribute 'Using' := '"Type": "Template", "URI": "E_BA_AC_SeqNumber_T"'}		 
	{attribute 'Description' := '"LCID": "1031", "Text": "Energie Rückgewinnung Zuluft Regler Temperatur"'}
	{attribute 'Description' := '"LCID": "1033", "Text": "Energy recovery Supply air controller temperature"'}
{endregion}
FUNCTION_BLOCK FB_BA_AC_ErcTSuACtrl EXTENDS FB_BA_View
VAR_INPUT
	bEn					: BOOL;
	fSpTSuA				: REAL;
	fTSuA				: REAL;
	bSync				: BOOL;
	fSync				: REAL;
	bDehumf				: BOOL;
	fTExtA				: REAL;
	fTWth				: REAL;
END_VAR
VAR_OUTPUT
	fY					: REAL;
	eAction				: E_BA_Action;
	bIsActive				: BOOL;	//	active sequence controller
	bSeqActv				: BOOL;	//	Release sequence link, sequence control is active	
END_VAR
VAR_IN_OUT
	stSeqLink			: ST_BA_SeqLink;	//	Sequenz Link Struktur	//	Sequence link structure	
END_VAR
VAR_INPUT CONSTANT PERSISTENT
	{attribute 'parameterCategory' := 'Behaviour'}
	fHysActionOn 		: REAL := 0.25;
	{attribute 'parameterCategory' := 'Behaviour'}
	fHysActionOff 		: REAL := -0.25;
END_VAR
VAR_INPUT CONSTANT
	Ctrl				: FB_BA_SeqCtrl;		 
END_VAR
VAR		
	HysAction			: FB_BA_Swi2P;
END_VAR

SUPER^(); // FB_BA_View
HysAction(bEn := TRUE, fIn := fTWth - fTExtA, fOn := fHysActionOn, fOff := fHysActionOff); // FB_BA_Swi2P
Ctrl(
    fSetpoint := fSpTSuA,
    fCtrlVal := fTSuA,
    eActionPgm := SEL(HysAction.bQ, E_BA_Action.eReverse, E_BA_Action.eDirect),
    bEnSync := bSync,
    fValSync := fSync,
    bEn := bEn AND NOT bDehumf,
    nMyNum := E_BA_AC_SeqNumber_T.eEnergyRecovery,
    stSeqLink := stSeqLink); // FB_BA_SeqCtrl
fY := Ctrl.fPresentValue;
bSeqActv := Ctrl.bSeqActv;
bIsActive := Ctrl.bIsActvSeqCtrl;
eAction := Ctrl.Actn;
fY := SEL(bEn AND bDehumf AND eAction = E_BA_Action.eDirect, Ctrl.fPresentValue, 100);

METHOD FB_init : BOOL
VAR_INPUT
	bInitRetains : BOOL; // if TRUE, the retain variables are initialized (warm start / cold start)
	bInCopyCode : BOOL;  // if TRUE, the instance afterwards gets moved into the copy code (online change)
END_VAR
Ctrl.iParent						:= THIS^;
Ctrl.iLabel							:= LblFun_LoopObject; 		
Ctrl.sObjectName					:= '{Idx=01}';						 
Ctrl.eOpMode						:= E_BA_PIDMode.ePID;								 	 										 
Ctrl.eOutputUnit					:= E_BA_Unit.eOther_Percent;
Ctrl.eActionRm						:= E_BA_Action.eReverse;
Ctrl.fProportionalConstant			:= 3;
Ctrl.fIntegralConstant				:= 180;
Ctrl.fDerivativeConstant			:= 0;
Ctrl.fMaxOutputRm 					:= 100;
Ctrl.fMinOutputRm					:= 0;
Ctrl.fCOVIncrement					:= 0;
Ctrl.nDampConstant					:= 0;
Ctrl.fNeutralZone					:= 0;
END_METHOD

END_FUNCTION_BLOCK

// ---- Templates/POUs/Trade/AirConditioning/Aggregates/PreHeater/FB_BA_AC_PreHtr.TcPOU
{region '#Template'}
	{attribute 'Version' := '5.1.0.1'}
	{attribute 'Tags' := '"LCID": "1031", "Text": "AC, Aggregates, pre-heater"'}
	{attribute 'Tags' := '"LCID": "1033", "Text": "AC, Aggregates, pre-heater"'}
	{attribute 'Using' := '"Type": "Template", "URI": "BA2_Param"'}
	{attribute 'Using' := '"Type": "Template", "URI": "EC_ID"'}
	{attribute 'Description' := '"LCID": "1031", "Text": "Aggregat Vorerhitzer"'}
	{attribute 'Description' := '"LCID": "1033", "Text": "Aggregate pre-heater"'}
{endregion}
FUNCTION_BLOCK FB_BA_AC_PreHtr EXTENDS FB_BA_View
VAR_INPUT
	fSpTSuA					: REAL;
	fTSuA					: REAL;
	bSyncTSuACtrl			: BOOL;
	fSyncTSuACtrl			: REAL;	
	bDehumf					: BOOL;
	bSkipPreRinse			: BOOL; // Vorspülen überspringen // Skip pre-rinse
	fTWth					: REAL;
	bTWthLowLimit			: BOOL;
	bResetDehumf    		: BOOL;
	stCmd					: ST_BA_Binary;				
END_VAR
VAR_OUTPUT
	bCmd					: BOOL;
	fPresentValue			: REAL;			
	bFrost					: BOOL;
	bPreRinseReady			: BOOL;  
	bActiveSeqCtrl			: BOOL;	
END_VAR
VAR_IN_OUT
	stTSeqLink				: ST_BA_SeqLink; // Sequenz Link Struktur // Sequence link structure	
END_VAR
VAR_INPUT CONSTANT PERSISTENT
	{attribute 'parameterCategory' := 'Behaviour'}
	fHysPuOn : REAL := 5.0;
	{attribute 'parameterCategory' := 'Behaviour'}
	fHysPuOff : REAL := 1.0;
END_VAR
VAR_INPUT CONSTANT
	TFl						: FB_BA_SensorAnalog;												
	TRt						: FB_BA_SensorAnalog;			
	TSuACtrl				: FB_BA_AC_PreHtrTSuACtrl;
	TRtCtrl					: FB_BA_AC_TRtCtrl;	
	TFrost					: FB_BA_SensorAnalog;																	
	TFrostPrtcCtrlAir		: FB_BA_PID_Sp;
	FrostThermostat			: FB_BA_SensorBinary;
	Vlv						: FB_BA_Vlv;
	Pu						: FB_BA_Pu1st;
	PlantLock				: FB_BA_PlantLock;																													 							
END_VAR
VAR
	bPrioSfty				: BOOL;
	bPrioCrit				: BOOL;		
	PrioSwiVal				: FB_BA_PrioSwi_B04;	
	
	HysPu					: FB_BA_Swi2P;
	SyncTSuACtrl			: FB_BA_RFTrig;
	SyncSeqCtrlIsActive		: FB_BA_RFTrig;
	PrioSwiSync				: FB_BA_PrioSwi_R04;	
END_VAR
VAR // added by the converter: edge detectors and wires of the graphical bodies
    _s1 : ST_BA_Analog;
    _s2 : ST_BA_Binary;
    _w1 : ANY;
    _w2 : BOOL;
END_VAR

SUPER^(); // FB_BA_View
PlantLock(); // FB_BA_PlantLock
bPrioSfty := PlantLock.bPrioHigh OR PlantLock.bPrioLocalHigh;
bPrioCrit := PlantLock.bPrioMedium OR PlantLock.bPrioLocalMedium;
TFl(); // FB_BA_SensorAnalog
TRt(); // FB_BA_SensorAnalog
PrioSwiVal(
    bEn01 := stCmd.bEnSfty,
    bVal01 := stCmd.bValSfty,
    bEn02 := stCmd.bEnCrit,
    bVal02 := stCmd.bValCrit,
    bEn03 := stCmd.bEnPgm,
    bVal03 := stCmd.bValPgm); // FB_BA_PrioSwi_B04
SyncTSuACtrl(bValue := bSyncTSuACtrl); // FB_BA_RFTrig
SyncSeqCtrlIsActive(bValue := TSuACtrl.bSeqActv); // FB_BA_RFTrig
PrioSwiSync(
    bEn01 := SyncTSuACtrl.Qr,
    fVal01 := fSyncTSuACtrl,
    bEn04 := SyncSeqCtrlIsActive.Qr AND bActiveSeqCtrl AND bTWthLowLimit,
    fVal04 := Vlv.fMdlt); // FB_BA_PrioSwi_R04
TSuACtrl(
    bEn := PrioSwiVal.bVal,
    fSpTSuA := fSpTSuA,
    fTSuA := fTSuA,
    bSync := PrioSwiSync.bQ,
    fSync := PrioSwiSync.fVal,
    bDehumf := bDehumf,
    bResetDehumf := bResetDehumf,
    stSeqLink := stTSeqLink); // FB_BA_AC_PreHtrTSuACtrl
bActiveSeqCtrl := TSuACtrl.bIsActive;
TRtCtrl(
    bEnPreRinse := PrioSwiVal.bVal,
    fTRt := TRt.fPresentValue,
    bTWthLowLimit := bTWthLowLimit,
    fTWth := fTWth,
    bSkipPreRinse := bSkipPreRinse,
    bSeqActive := stTSeqLink.bEnSeqLink); // FB_BA_AC_TRtCtrl
bPreRinseReady := TRtCtrl.bPreRinseReady;
TFrost(); // FB_BA_SensorAnalog
TFrostPrtcCtrlAir(bEn := TRUE, fX := TFrost.fPresentValue); // FB_BA_PID_Sp
FrostThermostat(); // FB_BA_SensorBinary
bFrost := TFrost.eEventState = E_BA_EventState.eLowLimit OR FrostThermostat.bPresentValue;
_w1 := MAX(TSuACtrl.fY, TRtCtrl.fY, TFrostPrtcCtrlAir.fY);
// compose _s1 : ST_BA_Analog
_s1.bEnSfty := stCmd.bEnSfty OR bPrioSfty;
_s1.fValSfty := _w1;
_s1.bEnCrit := stCmd.bEnCrit OR bPrioCrit OR bFrost;
_s1.fValCrit := SEL(bFrost, _w1, 100);
_s1.bEnPgm := TRUE;
_s1.fValPgm := _w1;
Vlv(stCmd := _s1); // FB_BA_Vlv
fPresentValue := Vlv.fMdlt;
HysPu(bEn := TRUE, fIn := fPresentValue, fOn := fHysPuOn, fOff := fHysPuOff); // FB_BA_Swi2P
_w2 := HysPu.bQ OR bTWthLowLimit OR bFrost;
// compose _s2 : ST_BA_Binary
_s2.bEnSfty := Vlv.stCmd.bEnSfty;
_s2.bValSfty := _w2;
_s2.bEnCrit := Vlv.stCmd.bEnCrit;
_s2.bValCrit := _w2;
_s2.bEnPgm := TRUE;
_s2.bValPgm := _w2;
Pu(stCmd := _s2); // FB_BA_Pu1st
bCmd := Pu.bCmd;

METHOD FB_init : BOOL
VAR_INPUT
	bInitRetains : BOOL; // if TRUE, the retain variables are initialized (warm start / cold start)
	bInCopyCode : BOOL;  // if TRUE, the instance afterwards gets moved into the copy code (online change)
END_VAR
PlantLock.Parent								:= THIS^;		

TFl.iParent										:= THIS^;		
TFl.iLabel										:= LblAgg_TemperatureFlow;   
TFl.sObjectName									:= '{Idx=11}';						 
TFl.eDPADMode									:= E_BA_DPADMode.eInclude;
TFl.MV.eUnit									:= E_BA_Unit.eTemperature_DegreesCelsius;
TFl.MV.fResolution 								:= 0.01;
TFl.MV.fScaleOffset 							:= 0; 
TFl.MV.bEventDetectionEnable					:= TRUE;
TFl.MV.eEnPlantLock								:= E_BA_LockPriority.eNoLock;
                            					                            					
TRt.iParent										:= THIS^;		
TRt.iLabel										:= LblAgg_TemperatureReturnFlow;   
TRt.sObjectName									:= '{Idx=11}';						 
TRt.eDPADMode									:= E_BA_DPADMode.eInclude;
TRt.MV.eUnit									:= E_BA_Unit.eTemperature_DegreesCelsius;
TRt.MV.fResolution 								:= 0.01;
TRt.MV.fScaleOffset 							:= 0;  
TRt.MV.bEventDetectionEnable					:= TRUE;
TRt.MV.eEnPlantLock								:= E_BA_LockPriority.eMedium;

TSuACtrl.iParent								:= THIS^;	
TSuACtrl.iLabel									:= LblCtl_SupplyAirTemperatureControl;   
TSuACtrl.sObjectName							:= '{Idx=11}';						 
TSuACtrl.eDPADMode								:= E_BA_DPADMode.eInclude;								

TRtCtrl.iParent									:= THIS^;
TRtCtrl.iLabel									:= LblCtl_ReturnWaterControl;   
TRtCtrl.sObjectName								:= '{Idx=12}';						 
TRtCtrl.eDPADMode								:= E_BA_DPADMode.eInclude;								
TRtCtrl.PreRinseDst.bEventDetectionEnable		:= TRUE;
TRtCtrl.PreRinseDst.eEnPlantLock				:= E_BA_LockPriority.eNoLock;
	                                				
TFrost.iParent									:= THIS^;		
TFrost.iLabel									:= LblCtl_TemperatureFrost;   
TFrost.sObjectName								:= '{Idx=11}';						 
TFrost.eDPADMode								:= E_BA_DPADMode.eInclude;
TFrost.MV.eUnit									:= E_BA_Unit.eTemperature_DegreesCelsius;
TFrost.MV.fResolution 							:= 0.0004577776;
TFrost.MV.fScaleOffset 							:= 0;  
TFrost.MV.bEventDetectionEnable					:= TRUE;
TFrost.MV.eEnPlantLock							:= E_BA_LockPriority.eMedium;

TFrostPrtcCtrlAir.iParent						:= THIS^;	
TFrostPrtcCtrlAir.iLabel						:= LblCtl_FrostProtectionControl;   
TFrostPrtcCtrlAir.sObjectName					:= '{Idx=13}';						 
TFrostPrtcCtrlAir.eDPADMode						:= E_BA_DPADMode.eInclude;
TFrostPrtcCtrlAir.Sp.fValueRm 					:= 5.0;
TFrostPrtcCtrlAir.Ctrl.fProportionalConstant	:= 5;
TFrostPrtcCtrlAir.Ctrl.fIntegralConstant		:= 60;	
TFrostPrtcCtrlAir.Ctrl.eActionRm				:= E_BA_Action.eReverse;

FrostThermostat.iParent							:= THIS^; 
FrostThermostat.iLabel							:= LblAgg_FrostProtectionMonitor;   
FrostThermostat.sObjectName						:= '{Idx=13}';						 
FrostThermostat.eDPADMode						:= E_BA_DPADMode.eInclude;
FrostThermostat.Input.iLabel					:= LblFun_OperationalMessage;   
FrostThermostat.Input.sObjectName				:= '{Idx=13}';						 
FrostThermostat.Input.ePolarity					:= E_BA_Polarity.eReverse;
FrostThermostat.Input.sActiveText 				:= txtEvent_Triggered;
FrostThermostat.Input.sInactiveText 			:= txtEvent_Normal;
FrostThermostat.Input.nEventClassID				:= EC_ID.NC30;
FrostThermostat.Input.aEventTransitionText[1]	:= txtEvent_Triggered;
FrostThermostat.Input.aEventTransitionText[2]	:= txtEvent_Error;
FrostThermostat.Input.aEventTransitionText[3]	:= txtEvent_Normal;
FrostThermostat.Input.bEventDetectionEnable		:= TRUE;
FrostThermostat.Input.eEnPlantLock				:= E_BA_LockPriority.eMedium;	

Vlv.iParent										:= THIS^;
Vlv.iLabel										:= LblAgg_Valve;    									 
Vlv.sObjectName									:= '{Idx=11}';						 
Vlv.eDPADMode									:= E_BA_DPADMode.eInclude;								
                            					
Pu.iParent										:= THIS^;
Pu.iLabel										:= LblAgg_Pump;   									 
Pu.sObjectName									:= '{Idx=11}';						 
Pu.eDPADMode									:= E_BA_DPADMode.eInclude;
Pu.Dst.bEventDetectionEnable					:= TRUE;
Pu.Dst.eEnPlantLock								:= E_BA_LockPriority.eMedium;
END_METHOD

END_FUNCTION_BLOCK

// ---- Templates/POUs/Universal/Sensor/FB_BA_SensorAnalog.TcPOU
{region '#Template'}
	{attribute 'Version' := '5.1.0.0'}
	{attribute 'Tags' := '"LCID": "1031", "Text": "Universal, Sensor, AI"'}
	{attribute 'Tags' := '"LCID": "1033", "Text": "Universal, Sensor, AI"'}
	{attribute 'Using' := '"Type": "Template", "URI": "EC_ID"'}
	{attribute 'Using' := '"Type": "Template", "URI": "BA2_Param"'}
	{attribute 'Description' := '"LCID": "1031", "Text": "AI mit IO"'}
	{attribute 'Description' := '"LCID": "1033", "Text": "AI with IO"'}
{endregion}
FUNCTION_BLOCK FB_BA_SensorAnalog EXTENDS FB_BA_View
VAR_INPUT
END_VAR
VAR_INPUT CONSTANT
	MV						: FB_BA_AI_Raw;		
END_VAR
VAR_OUTPUT
	fPresentValue			: REAL;
	bEvent					: BOOL;
	eEventState				: E_BA_EventState;	
END_VAR
VAR
END_VAR

SUPER^(); // FB_BA_View
MV(); // FB_BA_AI_Raw
bEvent := MV.bEvent;
eEventState := MV.eEventState;
fPresentValue := MV.fPresentValue;

METHOD FB_init : BOOL
VAR_INPUT
	bInitRetains : BOOL; // if TRUE, the retain variables are initialized (warm start / cold start)
	bInCopyCode : BOOL;  // if TRUE, the instance afterwards gets moved into the copy code (online change)
END_VAR
MV.iParent						:= THIS^;		
MV.iLabel						:= LblFun_MeasuredValue; 
MV.eUnit						:= E_BA_Unit.eTemperature_DegreesCelsius;
MV.fResolution 					:= 0.01;
MV.fScaleOffset 				:= 0; 	
MV.fCOVIncrement				:= BA2_Param.fDefCOVIncrement;
MV.nEventClassID				:= EC_ID.NC30;
MV.stTimeDelay.nToNormal		:= BA2_Param.nDefTimeDelay_ToNormal;
MV.stTimeDelay.nToAbnormal		:= BA2_Param.nDefTimeDelay_ToAbnormal;
MV.stHighLimit.bEnable			:= FALSE;
MV.stHighLimit.fValue			:= 0.0;		
MV.stLowLimit.bEnable			:= FALSE;
MV.stLowLimit.fValue			:= 0.0;
MV.fLimitDeadband 				:= BA2_Param.fDefLimitDeadband;
MV.aEventTransitionText[1]		:= txtEvent_Exceeded;
MV.aEventTransitionText[2]		:= txtEvent_Disturb;
MV.aEventTransitionText[3]		:= txtEvent_Normal;
MV.bEventDetectionEnable		:= TRUE;
MV.eEnPlantLock					:= E_BA_LockPriority.eNoLock;
END_METHOD

END_FUNCTION_BLOCK

// ---- Templates/POUs/Trade/AirConditioning/Aggregates/PreHeater/FB_BA_AC_PreHtrTSuACtrl.TcPOU
{region '#Template'}
	{attribute 'Version' := '5.0.1.0'}
	{attribute 'Tags' := '"LCID": "1031", "Text": "AC, Aggregates, Pre-heater, Temperature, Controller"'}
	{attribute 'Tags' := '"LCID": "1033", "Text": "AC, Aggregates, Pre-heater, Temperature, Controller"'}
	{attribute 'Using' := '"Type": "Template", "URI": "BA2_Param"'}
	{attribute 'Using' := '"Type": "Template", "URI": "EC_ID"'}
	{attribute 'Using' := '"Type": "Template", "URI": "E_BA_AC_SeqNumber_T"'}		 
	{attribute 'Description' := '"LCID": "1031", "Text": "Vorerhitzer Zuluft Regler Temperatur"'}
	{attribute 'Description' := '"LCID": "1033", "Text": "Pre-heater Supply air controller temperature"'}
{endregion}
FUNCTION_BLOCK FB_BA_AC_PreHtrTSuACtrl EXTENDS FB_BA_View
VAR_INPUT
	bEn						: BOOL;
	fSpTSuA					: REAL;
	fTSuA					: REAL;
	bSync					: BOOL;
	fSync					: REAL;
	bDehumf					: BOOL;
	bResetDehumf    		: BOOL;
END_VAR
VAR_OUTPUT
	fY              		: REAL;
	bIsActive				: BOOL;	//	active sequence controller
	bSeqActv				: BOOL;	//	Release sequence link, sequence control is active	
END_VAR
VAR_IN_OUT
	stSeqLink				: ST_BA_SeqLink;	//	Sequenz Link Struktur	//	Sequence link structure	
END_VAR
VAR_INPUT CONSTANT
	Ctrl					: FB_BA_SeqCtrl;	
END_VAR
VAR
	srDehumf				: SR;
	ftrigDeHum				: F_TRIG;
	rtrigSync				: R_TRIG;
	PrioSwiSync				: FB_BA_PrioSwi_R04;
END_VAR
VAR // added by the converter: edge detectors and wires of the graphical bodies
    _w1 : BOOL;
END_VAR

SUPER^(); // FB_BA_View
srDehumf(SET1 := bDehumf, RESET := bResetDehumf); // SR
_w1 := bEn AND NOT srDehumf.Q1 AND stSeqLink.bEnSeqLink;
ftrigDeHum(CLK := srDehumf.Q1); // F_TRIG
rtrigSync(CLK := bSync); // R_TRIG
PrioSwiSync(bEn02 := ftrigDeHum.Q, fVal02 := 0, bEn04 := rtrigSync.Q, fVal04 := fSync); // FB_BA_PrioSwi_R04
Ctrl(
    fSetpoint := fSpTSuA,
    fCtrlVal := fTSuA,
    eActionPgm := E_BA_Action.eReverse,
    bEnSync := PrioSwiSync.bQ,
    fValSync := PrioSwiSync.fVal,
    bEn := _w1,
    nMyNum := E_BA_AC_SeqNumber_T.ePreHeater,
    stSeqLink := stSeqLink); // FB_BA_SeqCtrl
fY := Ctrl.fPresentValue;
bSeqActv := Ctrl.bSeqActv;
bIsActive := Ctrl.bIsActvSeqCtrl;

METHOD FB_init : BOOL
VAR_INPUT
	bInitRetains : BOOL; // if TRUE, the retain variables are initialized (warm start / cold start)
	bInCopyCode : BOOL;  // if TRUE, the instance afterwards gets moved into the copy code (online change)
END_VAR
Ctrl.iParent						:= THIS^;
Ctrl.iLabel							:= LblFun_LoopObject; 		
Ctrl.sObjectName					:= '{Idx=01}';						 
Ctrl.eOpMode						:= E_BA_PIDMode.ePID;								 	 										 
Ctrl.eOutputUnit					:= E_BA_Unit.eOther_Percent;
Ctrl.fProportionalConstant			:= 3;
Ctrl.fIntegralConstant				:= 180;
Ctrl.fDerivativeConstant			:= 0;
Ctrl.fMaxOutputRm 					:= 100;
Ctrl.fMinOutputRm					:= 0;
Ctrl.fCOVIncrement					:= 0;
Ctrl.nDampConstant					:= 0;
Ctrl.fNeutralZone					:= 0;
END_METHOD

END_FUNCTION_BLOCK

// ---- Templates/POUs/Trade/AirConditioning/Aggregates/PreHeater/FB_BA_AC_TRtCtrl.TcPOU
{region '#Template'}
	{attribute 'Version' := '5.1.0.1'}
	{attribute 'Tags' := '"LCID": "1031", "Text": "AC, Aggregates, pre-heater, Return temperature control"'}
	{attribute 'Tags' := '"LCID": "1033", "Text": "AC, Aggregates, pre-heater, Return temperature control"'}
	{attribute 'Using' := '"Type": "Template", "URI": "BA2_Param"'}
	{attribute 'Using' := '"Type": "Template", "URI": "EC_ID"'}
	{attribute 'Description' := '"LCID": "1031", "Text": "Vorerhitzer Rücklauf Temperatur Regelung"'}
	{attribute 'Description' := '"LCID": "1033", "Text": "Pre-Heater return temperature control"'}
{endregion}
FUNCTION_BLOCK FB_BA_AC_TRtCtrl EXTENDS FB_BA_View
VAR_INPUT
	bEnPreRinse				: BOOL;
	fTRt					: REAL;
	bTWthLowLimit			: BOOL;// Außentemperatur unterer Grenzwert aktiv
	fTWth					: REAL;
	bSkipPreRinse			: BOOL; // Vorspülen überspringen // Skip pre-rinse
	bSeqActive				: BOOL;// Sequenz Regelung ist aktiv 	
END_VAR
VAR_OUTPUT
	fY						: REAL;
	bPreRinseActive			: BOOL;
	bPreRinseReady			: BOOL;
	bPreRinseDstb			: BOOL;
END_VAR
VAR_INPUT CONSTANT
	SpTRtW					: FB_BA_AV_Op;
	PreRinseDelay			: FB_BA_DlyOn;												 
	PreRinseDst				: FB_BA_BV;													   
	PreRinseSp				: FB_BA_Scale_02;																		
	Ctrl					: FB_BA_Loop;	
END_VAR
VAR
	rtrigPreRinse			: R_TRIG;
	rsPreRinseReady			: RS;
	rsPreRinseActive		: RS;
	PreRinseHys				: FB_BA_Swi2P;
END_VAR

SUPER^(); // FB_BA_View
SpTRtW(); // FB_BA_AV_Op
rtrigPreRinse(CLK := bEnPreRinse AND NOT bSkipPreRinse AND bTWthLowLimit); // R_TRIG
rsPreRinseActive(SET := rtrigPreRinse.Q, RESET1 := bSeqActive OR NOT bEnPreRinse OR bSkipPreRinse OR NOT bTWthLowLimit); // RS
bPreRinseActive := rsPreRinseActive.Q1;
PreRinseSp(fX := fTWth); // FB_BA_Scale_02
Ctrl(
    bEn := bTWthLowLimit,
    fSetpoint := SEL(rsPreRinseActive.Q1, SpTRtW.fPresentValue, PreRinseSp.fY),
    fCtrlVal := fTRt,
    eActionPgm := E_BA_Action.eReverse); // FB_BA_Loop
fY := Ctrl.fPresentValue;
PreRinseHys(
    bEn := bPreRinseActive AND BA2_Param.bDlyStartPLC,
    fIn := fTRt,
    fOn := PreRinseSp.fY,
    fOff := PreRinseSp.fY - 1); // FB_BA_Swi2P
rsPreRinseReady(SET := PreRinseHys.bQ OR PreRinseDelay.bQ, RESET1 := bSeqActive OR NOT bEnPreRinse); // RS
bPreRinseReady := rsPreRinseReady.Q1 OR bSkipPreRinse OR NOT bTWthLowLimit;
PreRinseDelay(bVal := bPreRinseActive AND NOT bPreRinseReady); // FB_BA_DlyOn
PreRinseDst(bEnPgm := TRUE, bValPgm := PreRinseDelay.bQ); // FB_BA_BV
bPreRinseDstb := PreRinseDst.bEvent;

METHOD FB_init : BOOL
VAR_INPUT
	bInitRetains : BOOL; // if TRUE, the retain variables are initialized (warm start / cold start)
	bInCopyCode : BOOL;  // if TRUE, the instance afterwards gets moved into the copy code (online change)
END_VAR
SpTRtW.iParent								:= THIS^;
SpTRtW.iLabel								:= LblFun_Setpoint; 
SpTRtW.sObjectName							:= '{Idx=01}';						 
SpTRtW.eUnit 								:= E_BA_Unit.eTemperature_DegreesCelsius;								 								
SpTRtW.fValueRm								:= 5.0;

PreRinseDelay.iParent						:= THIS^;	
PreRinseDelay.iLabel						:= LblCtl_DelayOn; 
PreRinseDelay.sObjectName					:= '{Idx=01}';						 
PreRinseDelay.eDPADMode						:= E_BA_DPADMode.eIncludeDescription;
PreRinseDelay.TiDly.iLabel					:= LblCtl_PreRinseDuration; 
PreRinseDelay.TiDly.sObjectName				:= '{Idx=01}';						 
PreRinseDelay.TiDly.fValueRm				:= 900;	

PreRinseDst.iParent							:= THIS^;
PreRinseDst.iLabel							:= LblCtl_DisturbancePreRinse; 
PreRinseDst.sObjectName						:= '{Idx=01}';						 
PreRinseDst.bEnOutOfService					:= FALSE;
PreRinseDst.sActiveText 					:= txtEvent_Triggered;
PreRinseDst.sInactiveText 					:= txtEvent_Normal;
PreRinseDst.nStateChangeCount				:= 0;
PreRinseDst.nActiveTimeElapsed				:= 0;
PreRinseDst.nMinimumOnTime					:= 0;
PreRinseDst.nMinimumOffTime					:= 0;
PreRinseDst.bEnManualRm						:= FALSE;	//	Priority  8	
PreRinseDst.bValManualRm					:= FALSE;	//	Priority  8
PreRinseDst.bDefaultValue					:= FALSE;
PreRinseDst.nEventClassID					:= EC_ID.NC30;
PreRinseDst.stTimeDelay.nToNormal			:= 0;
PreRinseDst.stTimeDelay.nToAbnormal			:= 0;
PreRinseDst.bAlarmValue						:= TRUE;
PreRinseDst.bAcknowledgeRm					:= FALSE;		
PreRinseDst.aEventTransitionText[1]			:= txtEvent_Triggered;
PreRinseDst.aEventTransitionText[2]			:= txtEvent_Error;
PreRinseDst.aEventTransitionText[3]			:= txtEvent_Normal;
PreRinseDst.bEventDetectionEnable			:= TRUE;
PreRinseDst.aEventEnable[1]					:= TRUE;			//	to_offnormal
PreRinseDst.aEventEnable[2]					:= FALSE;			//	to_fault
PreRinseDst.aEventEnable[3]					:= TRUE;			//	to_normal
PreRinseDst.eEnPlantLock					:= E_BA_LockPriority.eNoLock;	

PreRinseSp.iParent							:= THIS^;
PreRinseSp.iLabel							:= LblCtl_CalculationPreRinseSetpoint; 
PreRinseSp.sObjectName						:= '{Idx=02}';						 
PreRinseSp.eDPADMode						:= E_BA_DPADMode.eIncludeDescription;
PreRinseSp.X1.fValueRm						:= -10.0;
PreRinseSp.X2.fValueRm						:= 6.0;
PreRinseSp.Y1.fValueRm						:= 30.0;
PreRinseSp.Y2.fValueRm						:= 25.0;
PreRinseSp.YMin.fValueRm					:= 20.0;
PreRinseSp.YMax.fValueRm					:= 60.0;

Ctrl.iParent								:= THIS^;
Ctrl.iLabel									:= LblFun_LoopObject; 
Ctrl.sObjectName							:= '{Idx=01}';						 
Ctrl.eOpMode								:= E_BA_PIDMode.eP1ID;								 	 										 
Ctrl.eOutputUnit							:= E_BA_Unit.eOther_Percent;
Ctrl.eActionRm								:= E_BA_Action.eReverse;
Ctrl.fProportionalConstant					:= 3;
Ctrl.fIntegralConstant						:= 180;
Ctrl.fDerivativeConstant					:= 0;
Ctrl.fMaxOutputRm 							:= 100;
Ctrl.fMinOutputRm							:= 0;
Ctrl.fCOVIncrement							:= 0;
Ctrl.nDampConstant							:= 0;
Ctrl.fNeutralZone							:= 0;
END_METHOD

END_FUNCTION_BLOCK

// ---- Templates/POUs/Universal/Control/PID/FB_BA_PID_Sp.TcPOU
{region '#Template'}
	{attribute 'Version' := '5.0.0.0'}
	{attribute 'Tags' := '"LCID": "1031", "Text": "Universal, Control, PID, Loop"'}
	{attribute 'Tags' := '"LCID": "1033", "Text": "Universal, Control, PID, Loop"'}
	{attribute 'Using' := '"Type": "Template", "URI": "BA2_Param"'}
	{attribute 'Description' := '"LCID": "1031", "Text": "Regler mit Sollwert Object"'}
	{attribute 'Description' := '"LCID": "1033", "Text": "Controller with setpoint object"'}
{endregion}
FUNCTION_BLOCK FB_BA_PID_Sp EXTENDS FB_BA_View
VAR_INPUT
	bEn						: BOOL;
	fX						: REAL;
	bSync					: BOOL;
	fSync					: REAL;
END_VAR
VAR_OUTPUT
	fY						: REAL;
	fMax					: REAL;
	fMin					: REAL;	
END_VAR
VAR_INPUT CONSTANT
	Sp						: FB_BA_AV_Op;		 
	Ctrl					: FB_BA_Loop;	
END_VAR

SUPER^(); // FB_BA_View
Sp(); // FB_BA_AV_Op
Ctrl(bEn := bEn, fSetpoint := Sp.fPresentValue, fCtrlVal := fX, bEnSync := bSync, fValSync := fSync); // FB_BA_Loop
fY := Ctrl.fPresentValue;
fMin := Ctrl.fMinOutputRm;
fMax := Ctrl.fMaxOutputRm;

METHOD FB_init : BOOL
VAR_INPUT
	bInitRetains : BOOL; // if TRUE, the retain variables are initialized (warm start / cold start)
	bInCopyCode : BOOL;  // if TRUE, the instance afterwards gets moved into the copy code (online change)
END_VAR
Sp.iParent					:= THIS^;
Sp.iLabel					:= LblFun_Setpoint;   					 	 
Sp.eUnit 					:= E_BA_Unit.eTemperature_DegreesCelsius;								 
Sp.fValueRm					:= 21.0;															 
Sp.fCOVIncrement			:= BA2_Param.fDefCOVIncrement;

Ctrl.iParent				:= THIS^;
Ctrl.iLabel					:= LblFun_LoopObject;  
Ctrl.eOpMode				:= E_BA_PIDMode.ePID;								 	 										 
Ctrl.eOutputUnit			:= E_BA_Unit.eOther_Percent;
Ctrl.eActionRm				:= E_BA_Action.eReverse;
Ctrl.fProportionalConstant	:= 3;
Ctrl.fIntegralConstant		:= 180;
Ctrl.fDerivativeConstant	:= 0;
Ctrl.fMaxOutputRm 			:= 100;
Ctrl.fMinOutputRm			:= 0;
Ctrl.fCOVIncrement			:= 0;
Ctrl.nDampConstant			:= 0;
Ctrl.fNeutralZone			:= 0;
END_METHOD

END_FUNCTION_BLOCK

// ---- Templates/POUs/Universal/Sensor/FB_BA_SensorBinary.TcPOU
{region '#Template'}
	{attribute 'Version' := '5.1.0.0'}
	{attribute 'Tags' := '"LCID": "1031", "Text": "Universal, Sensor, BI"'}
	{attribute 'Tags' := '"LCID": "1033", "Text": "Universal, Sensor, BI"'}
	{attribute 'Using' := '"Type": "Template", "URI": "EC_ID"'}
	{attribute 'Using' := '"Type": "Template", "URI": "BA2_Param"'}
	{attribute 'Description' := '"LCID": "1031", "Text": "BI mit IO"'}
	{attribute 'Description' := '"LCID": "1033", "Text": "BI with IO"'}
{endregion}		 
FUNCTION_BLOCK FB_BA_SensorBinary EXTENDS FB_BA_View
VAR_INPUT
END_VAR
VAR_INPUT CONSTANT
	Input					: FB_BA_BI_Raw;		
END_VAR
VAR_OUTPUT
	bPresentValue			: BOOL;	
END_VAR
VAR
END_VAR

SUPER^(); // FB_BA_View
Input(); // FB_BA_BI_Raw
bPresentValue := Input.bPresentValue;

METHOD FB_init : BOOL
VAR_INPUT
	bInitRetains : BOOL; // if TRUE, the retain variables are initialized (warm start / cold start)
	bInCopyCode : BOOL;  // if TRUE, the instance afterwards gets moved into the copy code (online change)
END_VAR
Input.iParent						:= THIS^;
Input.iLabel						:= LblFun_Fault;
Input.ePolarity						:= E_BA_Polarity.eReverse;
Input.sActiveText 					:= txtEvent_Triggered;
Input.sInactiveText 				:= txtEvent_Normal;
Input.nEventClassID					:= EC_ID.NC30;
Input.stTimeDelay.nToNormal			:= BA2_Param.nDefTimeDelay_ToNormal;
Input.stTimeDelay.nToAbnormal		:= BA2_Param.nDefTimeDelay_ToAbnormal;
Input.bAlarmValue					:= TRUE;
Input.aEventTransitionText[1]		:= txtEvent_Triggered;
Input.aEventTransitionText[2]		:= txtEvent_Error;
Input.aEventTransitionText[3]		:= txtEvent_Normal;
Input.bEventDetectionEnable			:= TRUE;
Input.eEnPlantLock					:= E_BA_LockPriority.eNoLock;
END_METHOD

END_FUNCTION_BLOCK

// ---- Templates/POUs/Universal/Pump/1st/FB_BA_Pu1st.TcPOU
{region '#Template'}
	{attribute 'Version' := '5.0.0.0'}
	{attribute 'Tags' := '"LCID": "1031", "Text": "Universal, Pump"'}
	{attribute 'Tags' := '"LCID": "1033", "Text": "Universal, Pump"'}
	{attribute 'Using' := '"Type": "Template", "URI": "EC_ID"'}
	{attribute 'Using' := '"Type": "Template", "URI": "BA2_Param"'}
	{attribute 'Description' := '"LCID": "1031", "Text": "Pumpe 1 stufig"'}
	{attribute 'Description' := '"LCID": "1033", "Text": "Pump 1 stage"'}
{endregion}	 
FUNCTION_BLOCK FB_BA_Pu1st EXTENDS FB_BA_Mot1st
VAR_INPUT
	bAblkLock				: BOOL;	
END_VAR
VAR_INPUT CONSTANT
	DlyOff					: FB_BA_DlyOff;								
	Ablk					: FB_BA_AntiBlocking;							
END_VAR
VAR
	PrioSwiPgm				: FB_BA_PrioSwi_B04;
	tonAblkLock				: TON;
END_VAR
VAR // added by the converter: edge detectors and wires of the graphical bodies
    _s1 : ST_BA_Binary;
END_VAR

DlyOff(bVal := stCmd.bEnPgm AND stCmd.bValPgm); // FB_BA_DlyOff
tonAblkLock(IN := bAblkLock, PT := T#2s); // TON
Ablk(bFdb := bCmd, bLock := tonAblkLock.Q); // FB_BA_AntiBlocking
PrioSwiPgm(bEn03 := DlyOff.bQ, bVal03 := TRUE, bEn04 := Ablk.bQ, bVal04 := TRUE); // FB_BA_PrioSwi_B04
// compose _s1 : ST_BA_Binary
_s1.bEnSfty := stCmd.bEnSfty;
_s1.bValSfty := stCmd.bValSfty;
_s1.bEnCrit := stCmd.bEnCrit;
_s1.bValCrit := stCmd.bValCrit;
_s1.bEnPgm := PrioSwiPgm.bQ;
_s1.bValPgm := PrioSwiPgm.bVal;
SUPER^(stCmd := _s1); // FB_BA_Mot1st

METHOD FB_init : BOOL
VAR_INPUT
	bInitRetains : BOOL; // if TRUE, the retain variables are initialized (warm start / cold start)
	bInCopyCode : BOOL;  // if TRUE, the instance afterwards gets moved into the copy code (online change)
END_VAR
DlyOff.iParent			:= THIS^;	
DlyOff.iLabel			:= LblCtl_DelayOff;
DlyOff.eDPADMode		:= E_BA_DPADMode.eIncludeDescription;

Ablk.iParent			:= THIS^;	 
Ablk.iLabel				:= LblCtl_AntiBlocking;
Ablk.eDPADMode			:= E_BA_DPADMode.eIncludeDescription;
END_METHOD

END_FUNCTION_BLOCK

// ---- Templates/POUs/Universal/Control/TimeDelay/FB_BA_DlyOff.TcPOU
{region '#Template'}
	{attribute 'Version' := '5.0.0.0'}
	{attribute 'Tags' := '"LCID": "1031", "Text": "Universal, Control, Timer"'}
	{attribute 'Tags' := '"LCID": "1033", "Text": "Universal, Control, Timer"'}
	{attribute 'Using' := '"Type": "Template", "URI": "BA2_Param"'}
	{attribute 'Description' := '"LCID": "1031", "Text": "Zeitglied Ausschaltverzögert"'}
	{attribute 'Description' := '"LCID": "1033", "Text": "Timer switch-off delayed"'}
{endregion}
FUNCTION_BLOCK FB_BA_DlyOff EXTENDS FB_BA_View
VAR_INPUT
	bVal					: BOOL;	
END_VAR
VAR_OUTPUT
	bQ						: BOOL;	
	nRT						: UDINT;// Restzeit [s] // remaining time [s]
END_VAR
VAR_INPUT CONSTANT
	TiDly					: FB_BA_AV_Op;			
END_VAR	
VAR	
	tofDlyOff				: TOF;
END_VAR
VAR // added by the converter: edge detectors and wires of the graphical bodies
    _w1, _w2 : ANY;
END_VAR

SUPER^(); // FB_BA_View
TiDly(); // FB_BA_AV_Op
_w1 := F_BA_RealToTiSec(fSec := TiDly.fPresentValue);
tofDlyOff(IN := bVal, PT := _w1); // TOF
bQ := tofDlyOff.Q;
_w2 := F_BA_RemSecsTof(tofTimer := tofDlyOff);
nRT := _w2;

METHOD FB_init : BOOL
VAR_INPUT
	bInitRetains : BOOL; // if TRUE, the retain variables are initialized (warm start / cold start)
	bInCopyCode : BOOL;  // if TRUE, the instance afterwards gets moved into the copy code (online change)
END_VAR
TiDly.iParent			:= THIS^;
TiDly.iLabel			:= LblCtl_TimeDelay;
TiDly.eUnit 			:= E_BA_Unit.eTime_Seconds;								 
TiDly.fValueRm			:= 0;															 
TiDly.fCOVIncrement		:= BA2_Param.fDefCOVIncrement;
END_METHOD

END_FUNCTION_BLOCK

// ---- Templates/POUs/Trade/AirConditioning/General/FB_BA_AC_OpMod1St.TcPOU
{region '#Template'}
	{attribute 'Version' := '5.0.0.0'}
	{attribute 'Tags' := '"LCID": "1031", "Text": "AC, Allgemein, AHU, Betriebsart"'}
	{attribute 'Tags' := '"LCID": "1033", "Text": "AC, General, AHU, Operating mode"'}
	{attribute 'Using' := '"Type": "Template", "URI": "E_BA_AC_OpMod01"'}
	{attribute 'Using' := '"Type": "Template", "URI": "E_BA_OnOffA"'}
	{attribute 'Using' := '"Type": "Template", "URI": "E_BA_OnOff"'}
	{attribute 'Description' := '"LCID": "1031", "Text": "Betriebsart"'}
	{attribute 'Description' := '"LCID": "1033", "Text": "Operating mode"'}
{endregion}
FUNCTION_BLOCK FB_BA_AC_OpMod1St EXTENDS FB_BA_View
VAR_INPUT
	bSmExttSuA				: BOOL;	// smoke extraction supply air
	bSmExttExhA				: BOOL;	// smoke extraction exhaust air
	bFireDetc				: BOOL;	// fire detection alarm
	bForcVent				: BOOL;	// Forced ventilation
	bEmgOff					: BOOL;	// emergency stop
	bFrst					: BOOL;	// Frost protection is active
	bCentSwiOff				: BOOL;	// Central switch-off	
	bAlmShutOff				: BOOL;	// Shut Off plant collective alarm
	bNgtCol					: BOOL;	// Summer night cooling
	bColDwnPrtc				: BOOL;	// Cooling down protection
	bOvrHtgPrtc				: BOOL;	// Overheating protection
END_VAR
VAR_OUTPUT
	eOpMode					: E_BA_AC_OpMod01;
END_VAR
VAR_INPUT CONSTANT
	OpModMan				: FB_BA_MV_Op;	
	Sched					: FB_BA_SchedM;
	OpModPr					: FB_BA_MV_Op;
END_VAR
VAR
	PrioSwiOpMod			: FB_BA_PrioSwi_UDI24;
END_VAR

SUPER^(); // FB_BA_View
OpModMan(); // FB_BA_MV_Op
Sched(); // FB_BA_SchedM
PrioSwiOpMod(
    bEn02 := bSmExttSuA AND bSmExttExhA,
    nVal02 := E_BA_AC_OpMod01.eSmokeExtractionProgram,
    bEn03 := bSmExttSuA,
    nVal03 := E_BA_AC_OpMod01.eSmokeExtractionSupplyAir,
    bEn04 := bSmExttExhA,
    nVal04 := E_BA_AC_OpMod01.eSmokeExtractionExhaustAir,
    bEn05 := bFireDetc,
    nVal05 := E_BA_AC_OpMod01.eFire,
    bEn07 := bForcVent,
    nVal07 := E_BA_AC_OpMod01.eForcedVentilation,
    bEn08 := bEmgOff,
    nVal08 := E_BA_AC_OpMod01.eEmergency,
    bEn09 := bFrst,
    nVal09 := E_BA_AC_OpMod01.eFrost,
    bEn10 := bCentSwiOff,
    nVal10 := E_BA_AC_OpMod01.eCentralSwitchOff,
    bEn11 := bAlmShutOff,
    nVal11 := E_BA_AC_OpMod01.eAlarm,
    bEn14 := E_BA_OnOffA.eOff = OpModMan.nPresentValue,
    nVal14 := E_BA_AC_OpMod01.eOff,
    bEn15 := OpModMan.nPresentValue = E_BA_OnOffA.eOn,
    nVal15 := E_BA_AC_OpMod01.eOn,
    bEn18 := Sched.nPresentValue = E_BA_OnOff.eOn,
    nVal18 := E_BA_AC_OpMod01.eOn,
    bEn20 := bNgtCol,
    nVal20 := E_BA_AC_OpMod01.eNightCooling,
    bEn21 := bColDwnPrtc,
    nVal21 := E_BA_AC_OpMod01.eCoolDownProtection,
    bEn22 := bOvrHtgPrtc,
    nVal22 := E_BA_AC_OpMod01.eOverHeatingProtection,
    bEn24 := TRUE,
    nVal24 := E_BA_AC_OpMod01.eOFF); // FB_BA_PrioSwi_UDI24
OpModPr(nValuePgm := PrioSwiOpMod.nVal); // FB_BA_MV_Op
eOpMode := OpModPr.nPresentValue;

METHOD FB_init : BOOL
VAR_INPUT
	bInitRetains : BOOL; // if TRUE, the retain variables are initialized (warm start / cold start)
	bInCopyCode : BOOL;  // if TRUE, the instance afterwards gets moved into the copy code (online change)
END_VAR
OpModMan.iParent			:= THIS^;
OpModMan.iLabel				:= LblCtl_OperationModeSelection; 	
OpModMan.aStateText[1]		:= txtEvent_Auto;
OpModMan.aStateText[2]		:= txtEvent_Off;
OpModMan.aStateText[3]		:= txtEvent_On;
OpModMan.nValueRm			:= E_BA_OnOffA.eAutomatic;

OpModPr.iParent				:= THIS^;
OpModPr.iLabel				:= LblCtl_PresentOperationMode; 								 	 
OpModPr.aStateText[1]		:= txtEvent_Off;
OpModPr.aStateText[2]		:= txtEvent_On;
OpModPr.aStateText[3]		:= txtEvent_EmergencyStop;
OpModPr.aStateText[4]		:= txtEvent_Frost;
OpModPr.aStateText[5]		:= txtEvent_SmokeExtraction_P;
OpModPr.aStateText[6]		:= txtEvent_SmokeExtractionSupplyAir;
OpModPr.aStateText[7]		:= txtEvent_SmokeExtractionExtractAir;
OpModPr.aStateText[8]		:= txtEvent_Fire;
OpModPr.aStateText[9]		:= txtEvent_NightCooling;
OpModPr.aStateText[10]		:= txtEvent_CoolDownProtection;
OpModPr.aStateText[11]		:= txtEvent_OverHeatingProtection;
OpModPr.aStateText[12]		:= txtEvent_Disturb;
OpModPr.aStateText[13]		:= txtEvent_ForcedVentilation;
OpModPr.aStateText[14]		:= txtEvent_CentralSwitchOff; 		

Sched.iParent											:= THIS^;
Sched.iLabel											:= LblFun_Scheduler; 			
Sched.aStateText[1]										:= txtEvent_Off;
Sched.aStateText[2]										:= txtEvent_On;
Sched.nPredictTime										:= 0;
Sched.nDefaultValue										:= E_BA_OnOff.eOff;
Sched.bWriteWeekly										:= FALSE;
//	Monday
Sched.aWeek[E_BA_Weekday.eMonday,1].eState				:= E_BA_SchedEntryState.eValue;
Sched.aWeek[E_BA_Weekday.eMonday,1].uValue.udiVal		:= E_BA_OnOff.eOn;
Sched.aWeek[E_BA_Weekday.eMonday,1].stTime.nHour		:= 6;
Sched.aWeek[E_BA_Weekday.eMonday,1].stTime.nMinute		:= 0;
Sched.aWeek[E_BA_Weekday.eMonday,1].stTime.nSecond		:= 0;
Sched.aWeek[E_BA_Weekday.eMonday,2].eState				:= E_BA_SchedEntryState.eValue;
Sched.aWeek[E_BA_Weekday.eMonday,2].uValue.udiVal		:= E_BA_OnOff.eOff;
Sched.aWeek[E_BA_Weekday.eMonday,2].stTime.nHour		:= 20;
Sched.aWeek[E_BA_Weekday.eMonday,2].stTime.nMinute		:= 0;
Sched.aWeek[E_BA_Weekday.eMonday,2].stTime.nSecond		:= 0;
Sched.aWeek[E_BA_Weekday.eMonday,3].eState				:= E_BA_SchedEntryState.eValue;
Sched.aWeek[E_BA_Weekday.eMonday,3].uValue.udiVal		:= E_BA_OnOff.eOff;
Sched.aWeek[E_BA_Weekday.eMonday,3].stTime.nHour		:= 0;
Sched.aWeek[E_BA_Weekday.eMonday,3].stTime.nMinute		:= 0;
Sched.aWeek[E_BA_Weekday.eMonday,3].stTime.nSecond		:= 0;
//	Tuesday
Sched.aWeek[E_BA_Weekday.eTuesday,1].eState				:= E_BA_SchedEntryState.eValue;
Sched.aWeek[E_BA_Weekday.eTuesday,1].uValue.udiVal		:= E_BA_OnOff.eOn;
Sched.aWeek[E_BA_Weekday.eTuesday,1].stTime.nHour		:= 6;
Sched.aWeek[E_BA_Weekday.eTuesday,1].stTime.nMinute		:= 0;
Sched.aWeek[E_BA_Weekday.eTuesday,1].stTime.nSecond		:= 0;
Sched.aWeek[E_BA_Weekday.eTuesday,2].eState				:= E_BA_SchedEntryState.eValue;
Sched.aWeek[E_BA_Weekday.eTuesday,2].uValue.udiVal		:= E_BA_OnOff.eOff;
Sched.aWeek[E_BA_Weekday.eTuesday,2].stTime.nHour		:= 20;
Sched.aWeek[E_BA_Weekday.eTuesday,2].stTime.nMinute		:= 0;
Sched.aWeek[E_BA_Weekday.eTuesday,2].stTime.nSecond		:= 0;
Sched.aWeek[E_BA_Weekday.eTuesday,3].eState				:= E_BA_SchedEntryState.eValue;
Sched.aWeek[E_BA_Weekday.eTuesday,3].uValue.udiVal		:= E_BA_OnOff.eOff;
Sched.aWeek[E_BA_Weekday.eTuesday,3].stTime.nHour		:= 0;
Sched.aWeek[E_BA_Weekday.eTuesday,3].stTime.nMinute		:= 0;
Sched.aWeek[E_BA_Weekday.eTuesday,3].stTime.nSecond		:= 0;
//	Wednesday
Sched.aWeek[E_BA_Weekday.eWednesday,1].eState			:= E_BA_SchedEntryState.eValue;
Sched.aWeek[E_BA_Weekday.eWednesday,1].uValue.udiVal	:= E_BA_OnOff.eOn;
Sched.aWeek[E_BA_Weekday.eWednesday,1].stTime.nHour		:= 6;
Sched.aWeek[E_BA_Weekday.eWednesday,1].stTime.nMinute	:= 0;
Sched.aWeek[E_BA_Weekday.eWednesday,1].stTime.nSecond	:= 0;
Sched.aWeek[E_BA_Weekday.eWednesday,2].eState			:= E_BA_SchedEntryState.eValue;
Sched.aWeek[E_BA_Weekday.eWednesday,2].uValue.udiVal	:= E_BA_OnOff.eOff;
Sched.aWeek[E_BA_Weekday.eWednesday,2].stTime.nHour		:= 20;
Sched.aWeek[E_BA_Weekday.eWednesday,2].stTime.nMinute	:= 0;
Sched.aWeek[E_BA_Weekday.eWednesday,2].stTime.nSecond	:= 0;
Sched.aWeek[E_BA_Weekday.eWednesday,3].eState			:= E_BA_SchedEntryState.eValue;
Sched.aWeek[E_BA_Weekday.eWednesday,3].uValue.udiVal	:= E_BA_OnOff.eOff;
Sched.aWeek[E_BA_Weekday.eWednesday,3].stTime.nHour		:= 0;
Sched.aWeek[E_BA_Weekday.eWednesday,3].stTime.nMinute	:= 0;
Sched.aWeek[E_BA_Weekday.eWednesday,3].stTime.nSecond	:= 0;
//	Thursday
Sched.aWeek[E_BA_Weekday.eThursday,1].eState			:= E_BA_SchedEntryState.eValue;
Sched.aWeek[E_BA_Weekday.eThursday,1].uValue.udiVal		:= E_BA_OnOff.eOn;
Sched.aWeek[E_BA_Weekday.eThursday,1].stTime.nHour		:= 6;
Sched.aWeek[E_BA_Weekday.eThursday,1].stTime.nMinute	:= 0;
Sched.aWeek[E_BA_Weekday.eThursday,1].stTime.nSecond	:= 0;
Sched.aWeek[E_BA_Weekday.eThursday,2].eState			:= E_BA_SchedEntryState.eValue;
Sched.aWeek[E_BA_Weekday.eThursday,2].uValue.udiVal		:= E_BA_OnOff.eOff;
Sched.aWeek[E_BA_Weekday.eThursday,2].stTime.nHour		:= 20;
Sched.aWeek[E_BA_Weekday.eThursday,2].stTime.nMinute	:= 0;
Sched.aWeek[E_BA_Weekday.eThursday,2].stTime.nSecond	:= 0;
Sched.aWeek[E_BA_Weekday.eThursday,3].eState			:= E_BA_SchedEntryState.eValue;
Sched.aWeek[E_BA_Weekday.eThursday,3].uValue.udiVal		:= E_BA_OnOff.eOff;
Sched.aWeek[E_BA_Weekday.eThursday,3].stTime.nHour		:= 0;
Sched.aWeek[E_BA_Weekday.eThursday,3].stTime.nMinute	:= 0;
Sched.aWeek[E_BA_Weekday.eThursday,3].stTime.nSecond	:= 0;
//	Friday
Sched.aWeek[E_BA_Weekday.eFriday,1].eState				:= E_BA_SchedEntryState.eValue;
Sched.aWeek[E_BA_Weekday.eFriday,1].uValue.udiVal		:= E_BA_OnOff.eOn;
Sched.aWeek[E_BA_Weekday.eFriday,1].stTime.nHour		:= 6;
Sched.aWeek[E_BA_Weekday.eFriday,1].stTime.nMinute		:= 0;
Sched.aWeek[E_BA_Weekday.eFriday,1].stTime.nSecond		:= 0;
Sched.aWeek[E_BA_Weekday.eFriday,2].eState				:= E_BA_SchedEntryState.eValue;
Sched.aWeek[E_BA_Weekday.eFriday,2].uValue.udiVal		:= E_BA_OnOff.eOff;
Sched.aWeek[E_BA_Weekday.eFriday,2].stTime.nHour		:= 20;
Sched.aWeek[E_BA_Weekday.eFriday,2].stTime.nMinute		:= 0;
Sched.aWeek[E_BA_Weekday.eFriday,2].stTime.nSecond		:= 0;
Sched.aWeek[E_BA_Weekday.eFriday,3].eState				:= E_BA_SchedEntryState.eValue;
Sched.aWeek[E_BA_Weekday.eFriday,3].uValue.udiVal		:= E_BA_OnOff.eOff;
Sched.aWeek[E_BA_Weekday.eFriday,3].stTime.nHour		:= 0;
Sched.aWeek[E_BA_Weekday.eFriday,3].stTime.nMinute		:= 0;
Sched.aWeek[E_BA_Weekday.eFriday,3].stTime.nSecond		:= 0;
Sched.bWriteException									:= FALSE;
END_METHOD

END_FUNCTION_BLOCK

// ---- Templates/POUs/Trade/AirConditioning/General/FB_BA_AC_OpModAggBinary.TcPOU
{region '#Template'}
	{attribute 'Version' := '5.0.0.0'}
	{attribute 'Tags' := '"LCID": "1031", "Text": "AC, Allgemein, AHU, Betriebsart"'}
	{attribute 'Tags' := '"LCID": "1033", "Text": "AC, General, AHU, Operating mode"'}
	{attribute 'Using' := '"Type": "Template", "URI": "E_BA_AC_OpMod01"'}
	{attribute 'Description' := '"LCID": "1031", "Text": "Betriebsart"'}
	{attribute 'Description' := '"LCID": "1033", "Text": "Operating mode"'}
{endregion}

FUNCTION_BLOCK FB_BA_AC_OpModAggBinary
VAR_INPUT
	eOpMode					: E_BA_AC_OpMod01;
	bFdb					: BOOL;
	fDlyOn					: REAL;	
	fDlyOff					: REAL;	
END_VAR
VAR_OUTPUT
	bVal					: BOOL;	
	_bFdb					: BOOL;	
	nDelayOn				: UDINT;
	nDelayOff				: UDINT;
END_VAR
VAR_INPUT CONSTANT
	OpModVal				: FB_BA_MMUX_B16;
	DelayOn					: FB_BA_MMUX_B16;
	DelayOff				: FB_BA_MMUX_B16;
	IgnoreFdb				: FB_BA_MMUX_B16;	
END_VAR
VAR_INPUT CONSTANT PERSISTENT
	bInit					: BOOL := TRUE;
	arrOpModVal				: ARRAY [1..16] OF BOOL;
	arrIgnoreDelayOnVal 	: ARRAY [1..16] OF BOOL;
	arrIgnoreDelayOffVal	: ARRAY [1..16] OF BOOL;
	arrIgnoreFdbVal 		: ARRAY [1..16] OF BOOL;	
END_VAR
VAR // added by the converter: edge detectors and wires of the graphical bodies
    _w1, _w2 : UDINT;
END_VAR

